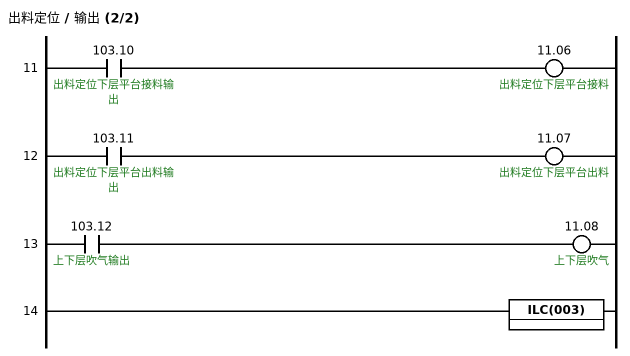
; rung 11
LD 103.10  ; 出料定位下层平台接料输出
OUT 11.06  ; 出料定位下层平台接料
; rung 12
LD 103.11  ; 出料定位下层平台出料输出
OUT 11.07  ; 出料定位下层平台出料
; rung 13
LD 103.12  ; 上下层吹气输出
OUT 11.08  ; 上下层吹气
; rung 14
ILC(003)

### Section END
; rung 0
END(001)

## Program 进出料转移 (cyclic task 3)

### Section Main

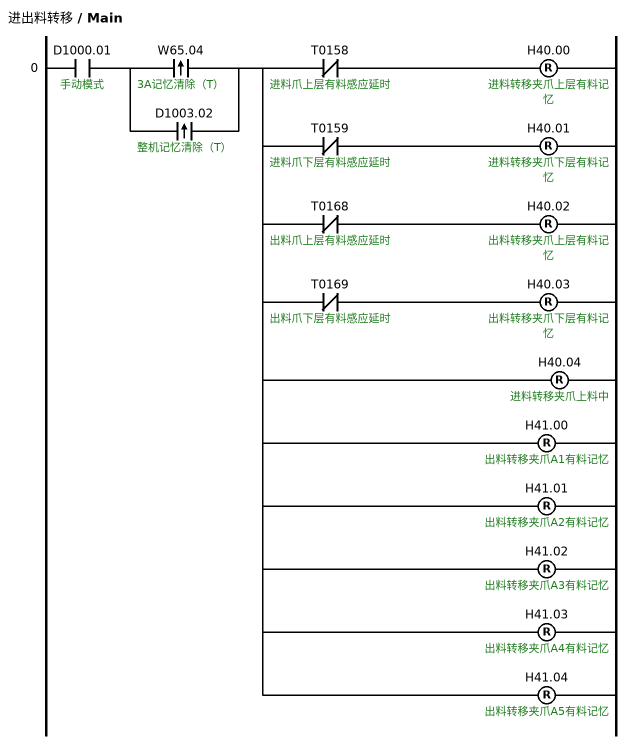
; rung 0
LD D1000.01  ; 手动模式
@LD W65.04  ; 3A记忆清除（T）
@OR D1003.02  ; 整机记忆清除（T）
ANDLD
OUT TR0
ANDNOT T0158  ; 进料爪上层有料感应延时
RSET H40.00  ; 进料转移夹爪上层有料记忆
LD TR0
ANDNOT T0159  ; 进料爪下层有料感应延时
RSET H40.01  ; 进料转移夹爪下层有料记忆
LD TR0
ANDNOT T0168  ; 出料爪上层有料感应延时
RSET H40.02  ; 出料转移夹爪上层有料记忆
LD TR0
ANDNOT T0169  ; 出料爪下层有料感应延时
RSET H40.03  ; 出料转移夹爪下层有料记忆
LD TR0
RSET H40.04  ; 进料转移夹爪上料中
RSET H41.00  ; 出料转移夹爪A1有料记忆
RSET H41.01  ; 出料转移夹爪A2有料记忆
RSET H41.02  ; 出料转移夹爪A3有料记忆
RSET H41.03  ; 出料转移夹爪A4有料记忆
RSET H41.04  ; 出料转移夹爪A5有料记忆

### Section _3ST进出料转移

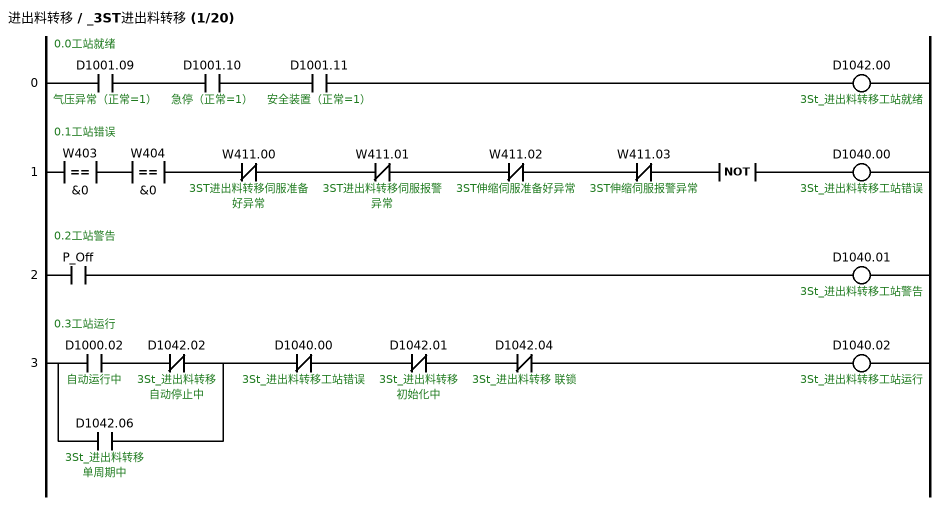
; rung 0: 0.0工站就绪
LD D1001.09  ; 气压异常（正常=1）
AND D1001.10  ; 急停（正常=1）
AND D1001.11  ; 安全装置（正常=1）
OUT D1042.00  ; 3St_进出料转移工站就绪
; rung 1: 0.1工站错误
LD=(300) W403 &0
AND=(300) W404 &0
ANDNOT W411.00  ; 3ST进出料转移伺服准备好异常
ANDNOT W411.01  ; 3ST进出料转移伺服报警异常
ANDNOT W411.02  ; 3ST伸缩伺服准备好异常
ANDNOT W411.03  ; 3ST伸缩伺服报警异常
NOT(520)
OUT D1040.00  ; 3St_进出料转移工站错误
; rung 2: 0.2工站警告
LD P_Off
OUT D1040.01  ; 3St_进出料转移工站警告
; rung 3: 0.3工站运行
LD D1000.02  ; 自动运行中
ANDNOT D1042.02  ; 3St_进出料转移 自动停止中
OR D1042.06  ; 3St_进出料转移 单周期中
ANDNOT D1040.00  ; 3St_进出料转移工站错误
ANDNOT D1042.01  ; 3St_进出料转移 初始化中
ANDNOT D1042.04  ; 3St_进出料转移 联锁
OUT D1040.02  ; 3St_进出料转移工站运行

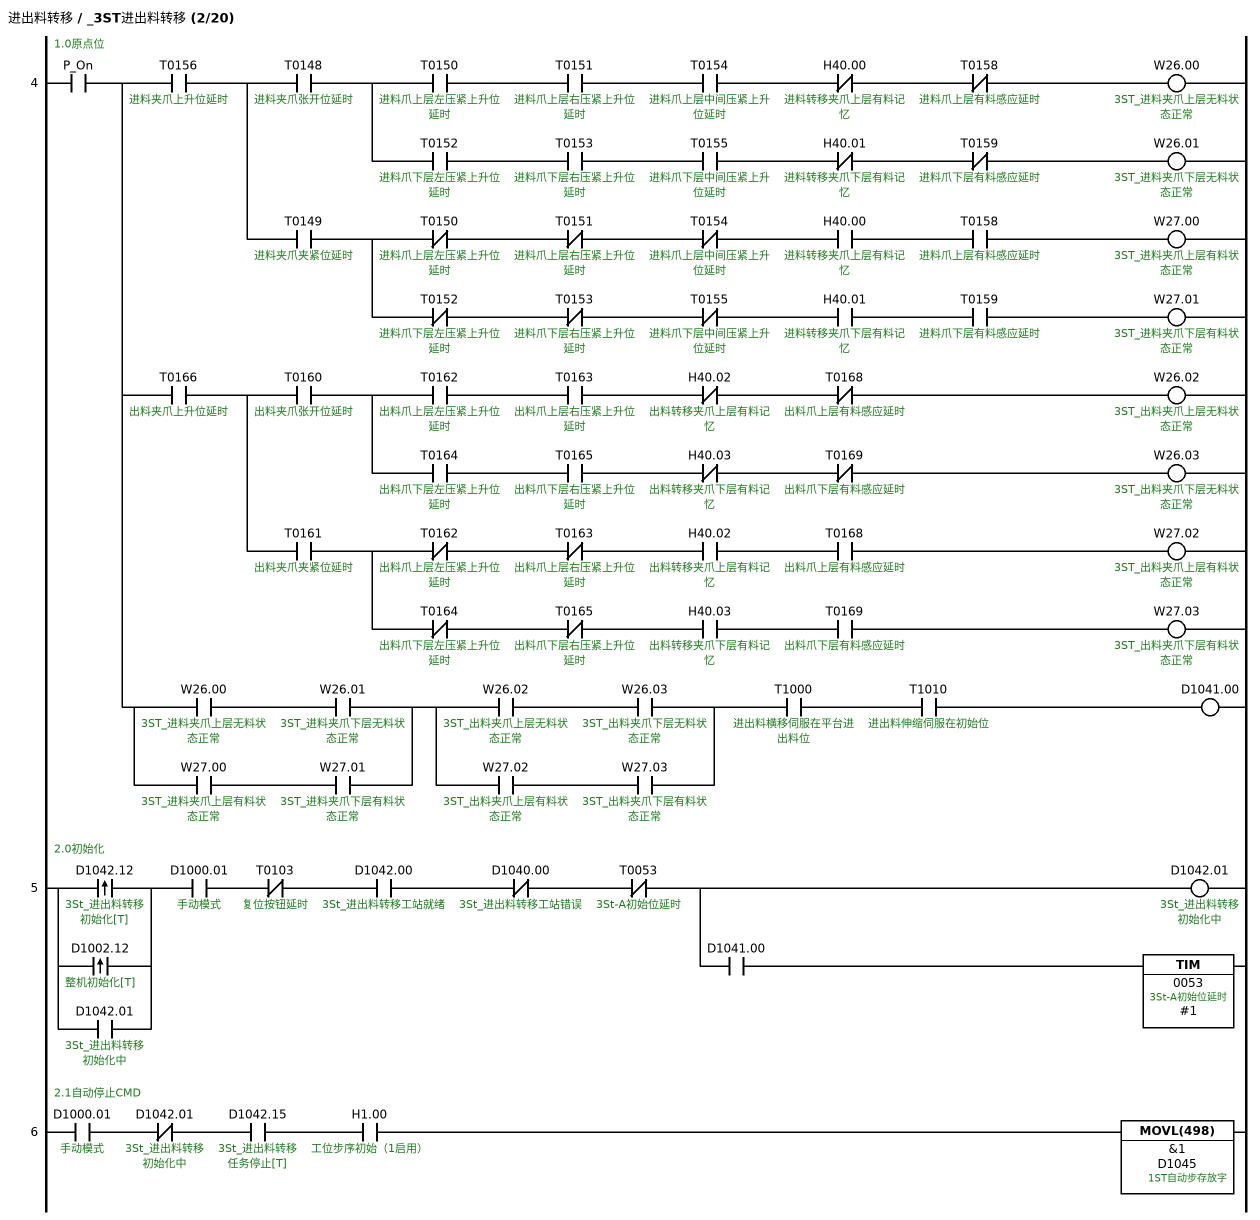
; rung 4: 1.0原点位
LD P_On
OUT TR0
AND T0156  ; 进料夹爪上升位延时
OUT TR1
AND T0148  ; 进料夹爪张开位延时
OUT TR2
AND T0150  ; 进料爪上层左压紧上升位延时
AND T0151  ; 进料爪上层右压紧上升位延时
AND T0154  ; 进料爪上层中间压紧上升位延时
ANDNOT H40.00  ; 进料转移夹爪上层有料记忆
ANDNOT T0158  ; 进料爪上层有料感应延时
OUT W26.00  ; 3ST_进料夹爪上层无料状态正常
LD TR2
AND T0152  ; 进料爪下层左压紧上升位延时
AND T0153  ; 进料爪下层右压紧上升位延时
AND T0155  ; 进料爪下层中间压紧上升位延时
ANDNOT H40.01  ; 进料转移夹爪下层有料记忆
ANDNOT T0159  ; 进料爪下层有料感应延时
OUT W26.01  ; 3ST_进料夹爪下层无料状态正常
LD TR1
AND T0149  ; 进料夹爪夹紧位延时
OUT TR1
ANDNOT T0150  ; 进料爪上层左压紧上升位延时
ANDNOT T0151  ; 进料爪上层右压紧上升位延时
ANDNOT T0154  ; 进料爪上层中间压紧上升位延时
AND H40.00  ; 进料转移夹爪上层有料记忆
AND T0158  ; 进料爪上层有料感应延时
OUT W27.00  ; 3ST_进料夹爪上层有料状态正常
LD TR1
ANDNOT T0152  ; 进料爪下层左压紧上升位延时
ANDNOT T0153  ; 进料爪下层右压紧上升位延时
ANDNOT T0155  ; 进料爪下层中间压紧上升位延时
AND H40.01  ; 进料转移夹爪下层有料记忆
AND T0159  ; 进料爪下层有料感应延时
OUT W27.01  ; 3ST_进料夹爪下层有料状态正常
LD TR0
AND T0166  ; 出料夹爪上升位延时
OUT TR1
AND T0160  ; 出料夹爪张开位延时
OUT TR2
AND T0162  ; 出料爪上层左压紧上升位延时
AND T0163  ; 出料爪上层右压紧上升位延时
ANDNOT H40.02  ; 出料转移夹爪上层有料记忆
ANDNOT T0168  ; 出料爪上层有料感应延时
OUT W26.02  ; 3ST_出料夹爪上层无料状态正常
LD TR2
AND T0164  ; 出料爪下层左压紧上升位延时
AND T0165  ; 出料爪下层右压紧上升位延时
ANDNOT H40.03  ; 出料转移夹爪下层有料记忆
ANDNOT T0169  ; 出料爪下层有料感应延时
OUT W26.03  ; 3ST_出料夹爪下层无料状态正常
LD TR1
AND T0161  ; 出料夹爪夹紧位延时
OUT TR1
ANDNOT T0162  ; 出料爪上层左压紧上升位延时
ANDNOT T0163  ; 出料爪上层右压紧上升位延时
AND H40.02  ; 出料转移夹爪上层有料记忆
AND T0168  ; 出料爪上层有料感应延时
OUT W27.02  ; 3ST_出料夹爪上层有料状态正常
LD TR1
ANDNOT T0164  ; 出料爪下层左压紧上升位延时
ANDNOT T0165  ; 出料爪下层右压紧上升位延时
AND H40.03  ; 出料转移夹爪下层有料记忆
AND T0169  ; 出料爪下层有料感应延时
OUT W27.03  ; 3ST_出料夹爪下层有料状态正常
LD TR0
LD W26.00  ; 3ST_进料夹爪上层无料状态正常
AND W26.01  ; 3ST_进料夹爪下层无料状态正常
LD W27.00  ; 3ST_进料夹爪上层有料状态正常
AND W27.01  ; 3ST_进料夹爪下层有料状态正常
ORLD
ANDLD
LD W26.02  ; 3ST_出料夹爪上层无料状态正常
AND W26.03  ; 3ST_出料夹爪下层无料状态正常
LD W27.02  ; 3ST_出料夹爪上层有料状态正常
AND W27.03  ; 3ST_出料夹爪下层有料状态正常
ORLD
ANDLD
AND T1000  ; 进出料横移伺服在平台进出料位
AND T1010  ; 进出料伸缩伺服在初始位
OUT D1041.00
; rung 5: 2.0初始化
@LD D1042.12  ; 3St_进出料转移 初始化[T]
@OR D1002.12  ; 整机初始化[T]
OR D1042.01  ; 3St_进出料转移 初始化中
AND D1000.01  ; 手动模式
ANDNOT T0103  ; 复位按钮延时
AND D1042.00  ; 3St_进出料转移工站就绪
ANDNOT D1040.00  ; 3St_进出料转移工站错误
ANDNOT T0053  ; 3St-A初始位延时
OUT D1042.01  ; 3St_进出料转移 初始化中
AND D1041.00
TIM 0053 #1  ; 3St-A初始位延时
; rung 6: 2.1自动停止CMD
LD D1000.01  ; 手动模式
ANDNOT D1042.01  ; 3St_进出料转移 初始化中
AND D1042.15  ; 3St_进出料转移 任务停止[T]
AND H1.00  ; 工位步序初始（1启用）
MOVL(498) &1 D1045  ; 1ST自动步存放字

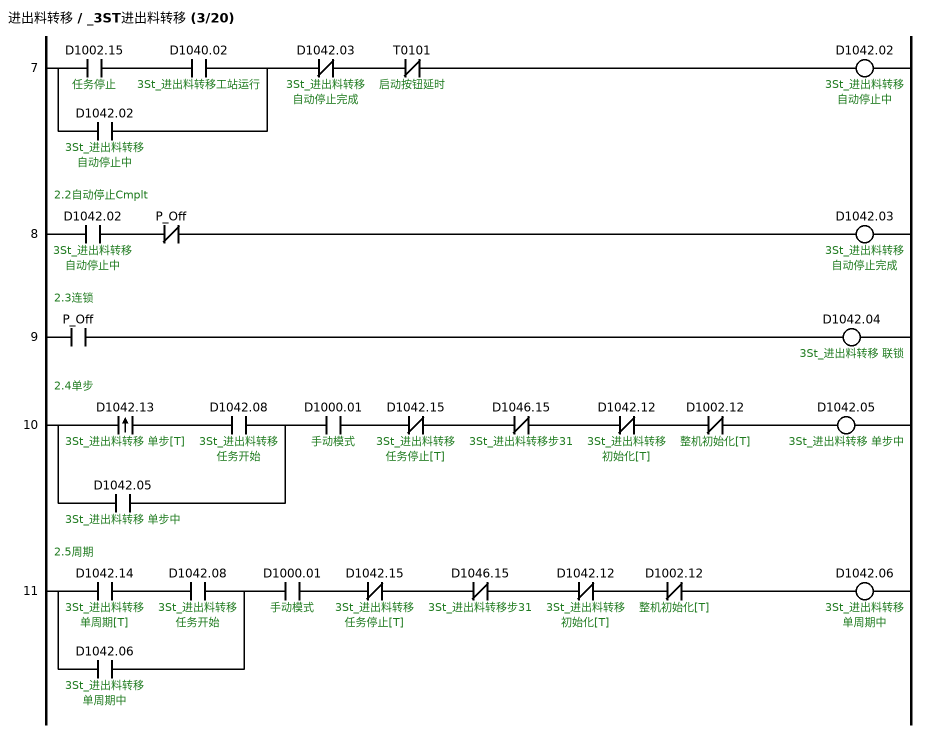
; rung 7
LD D1002.15  ; 任务停止
AND D1040.02  ; 3St_进出料转移工站运行
OR D1042.02  ; 3St_进出料转移 自动停止中
ANDNOT D1042.03  ; 3St_进出料转移 自动停止完成
ANDNOT T0101  ; 启动按钮延时
OUT D1042.02  ; 3St_进出料转移 自动停止中
; rung 8: 2.2自动停止Cmplt
LD D1042.02  ; 3St_进出料转移 自动停止中
ANDNOT P_Off
OUT D1042.03  ; 3St_进出料转移 自动停止完成
; rung 9: 2.3连锁
LD P_Off
OUT D1042.04  ; 3St_进出料转移 联锁
; rung 10: 2.4单步
@LD D1042.13  ; 3St_进出料转移 单步[T]
AND D1042.08  ; 3St_进出料转移 任务开始
OR D1042.05  ; 3St_进出料转移 单步中
AND D1000.01  ; 手动模式
ANDNOT D1042.15  ; 3St_进出料转移 任务停止[T]
ANDNOT D1046.15  ; 3St_进出料转移步31
ANDNOT D1042.12  ; 3St_进出料转移 初始化[T]
ANDNOT D1002.12  ; 整机初始化[T]
OUT D1042.05  ; 3St_进出料转移 单步中
; rung 11: 2.5周期
LD D1042.14  ; 3St_进出料转移 单周期[T]
AND D1042.08  ; 3St_进出料转移 任务开始
OR D1042.06  ; 3St_进出料转移 单周期中
AND D1000.01  ; 手动模式
ANDNOT D1042.15  ; 3St_进出料转移 任务停止[T]
ANDNOT D1046.15  ; 3St_进出料转移步31
ANDNOT D1042.12  ; 3St_进出料转移 初始化[T]
ANDNOT D1002.12  ; 整机初始化[T]
OUT D1042.06  ; 3St_进出料转移 单周期中

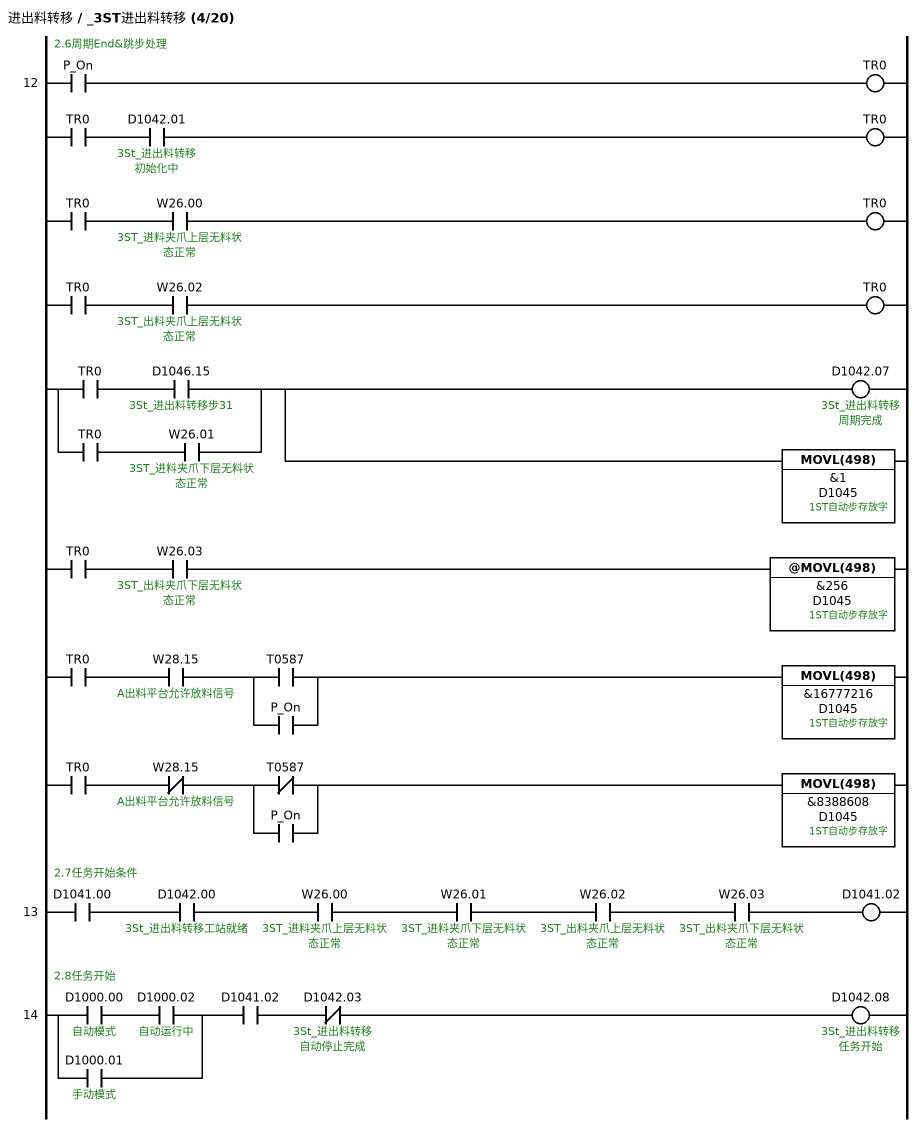
; rung 12: 2.6周期End&跳步处理
LD P_On
OUT TR0
AND D1046.15  ; 3St_进出料转移步31
LD TR0
AND D1042.01  ; 3St_进出料转移 初始化中
OUT TR0
AND W26.01  ; 3ST_进料夹爪下层无料状态正常
ORLD
OUT D1042.07  ; 3St_进出料转移 周期完成
MOVL(498) &1 D1045  ; 1ST自动步存放字
LD TR0
AND W26.00  ; 3ST_进料夹爪上层无料状态正常
OUT TR0
AND W26.03  ; 3ST_出料夹爪下层无料状态正常
@MOVL(498) &256 D1045  ; 1ST自动步存放字  // D1045.08  3ST_A到进料等待位
LD TR0
AND W26.02  ; 3ST_出料夹爪上层无料状态正常
OUT TR0
AND W28.15  ; A出料平台允许放料信号
LD T0587
OR P_On
ANDLD
MOVL(498) &16777216 D1045  ; 1ST自动步存放字  // D1046.08  3ST_A到出料位出料/夹爪下降
LD TR0
ANDNOT W28.15  ; A出料平台允许放料信号
LDNOT T0587
OR P_On
ANDLD
MOVL(498) &8388608 D1045  ; 1ST自动步存放字  // D1046.07  3ST_A到出料等待位
; rung 13: 2.7任务开始条件
LD D1041.00
AND D1042.00  ; 3St_进出料转移工站就绪
AND W26.00  ; 3ST_进料夹爪上层无料状态正常
AND W26.01  ; 3ST_进料夹爪下层无料状态正常
AND W26.02  ; 3ST_出料夹爪上层无料状态正常
AND W26.03  ; 3ST_出料夹爪下层无料状态正常
OUT D1041.02
; rung 14: 2.8任务开始
LD D1000.00  ; 自动模式
AND D1000.02  ; 自动运行中
OR D1000.01  ; 手动模式
AND D1041.02
ANDNOT D1042.03  ; 3St_进出料转移 自动停止完成
OUT D1042.08  ; 3St_进出料转移 任务开始

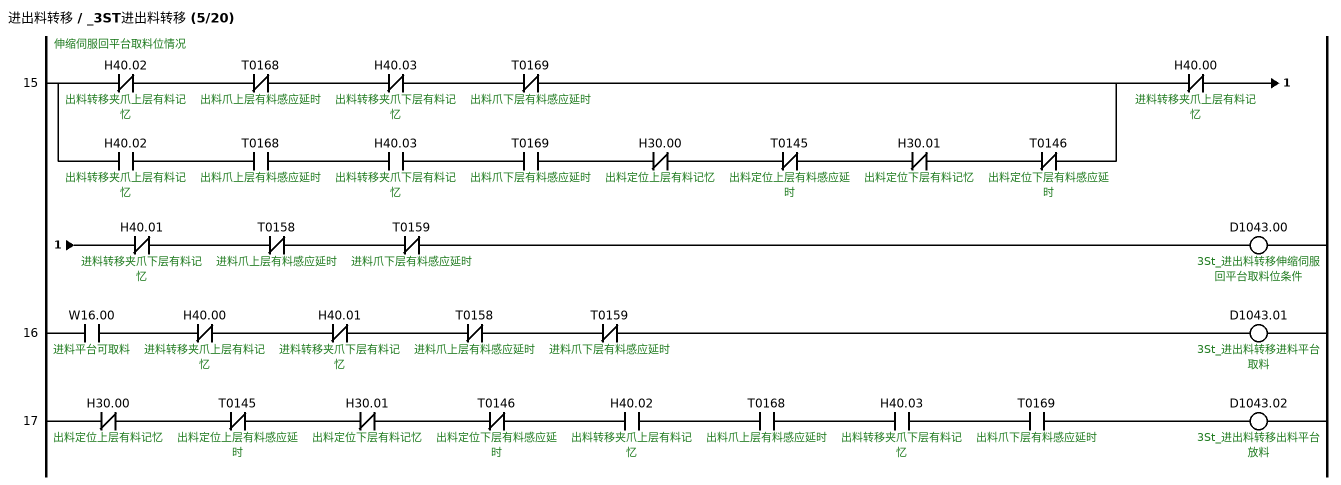
; rung 15: 伸缩伺服回平台取料位情况
LDNOT H40.02  ; 出料转移夹爪上层有料记忆
ANDNOT T0168  ; 出料爪上层有料感应延时
ANDNOT H40.03  ; 出料转移夹爪下层有料记忆
ANDNOT T0169  ; 出料爪下层有料感应延时
LD H40.02  ; 出料转移夹爪上层有料记忆
AND T0168  ; 出料爪上层有料感应延时
AND H40.03  ; 出料转移夹爪下层有料记忆
AND T0169  ; 出料爪下层有料感应延时
ANDNOT H30.00  ; 出料定位上层有料记忆
ANDNOT T0145  ; 出料定位上层有料感应延时
ANDNOT H30.01  ; 出料定位下层有料记忆
ANDNOT T0146  ; 出料定位下层有料感应延时
ORLD
ANDNOT H40.00  ; 进料转移夹爪上层有料记忆
ANDNOT H40.01  ; 进料转移夹爪下层有料记忆
ANDNOT T0158  ; 进料爪上层有料感应延时
ANDNOT T0159  ; 进料爪下层有料感应延时
OUT D1043.00  ; 3St_进出料转移伸缩伺服回平台取料位条件
; rung 16
LD W16.00  ; 进料平台可取料
ANDNOT H40.00  ; 进料转移夹爪上层有料记忆
ANDNOT H40.01  ; 进料转移夹爪下层有料记忆
ANDNOT T0158  ; 进料爪上层有料感应延时
ANDNOT T0159  ; 进料爪下层有料感应延时
OUT D1043.01  ; 3St_进出料转移进料平台取料
; rung 17
LDNOT H30.00  ; 出料定位上层有料记忆
ANDNOT T0145  ; 出料定位上层有料感应延时
ANDNOT H30.01  ; 出料定位下层有料记忆
ANDNOT T0146  ; 出料定位下层有料感应延时
AND H40.02  ; 出料转移夹爪上层有料记忆
AND T0168  ; 出料爪上层有料感应延时
AND H40.03  ; 出料转移夹爪下层有料记忆
AND T0169  ; 出料爪下层有料感应延时
OUT D1043.02  ; 3St_进出料转移出料平台放料

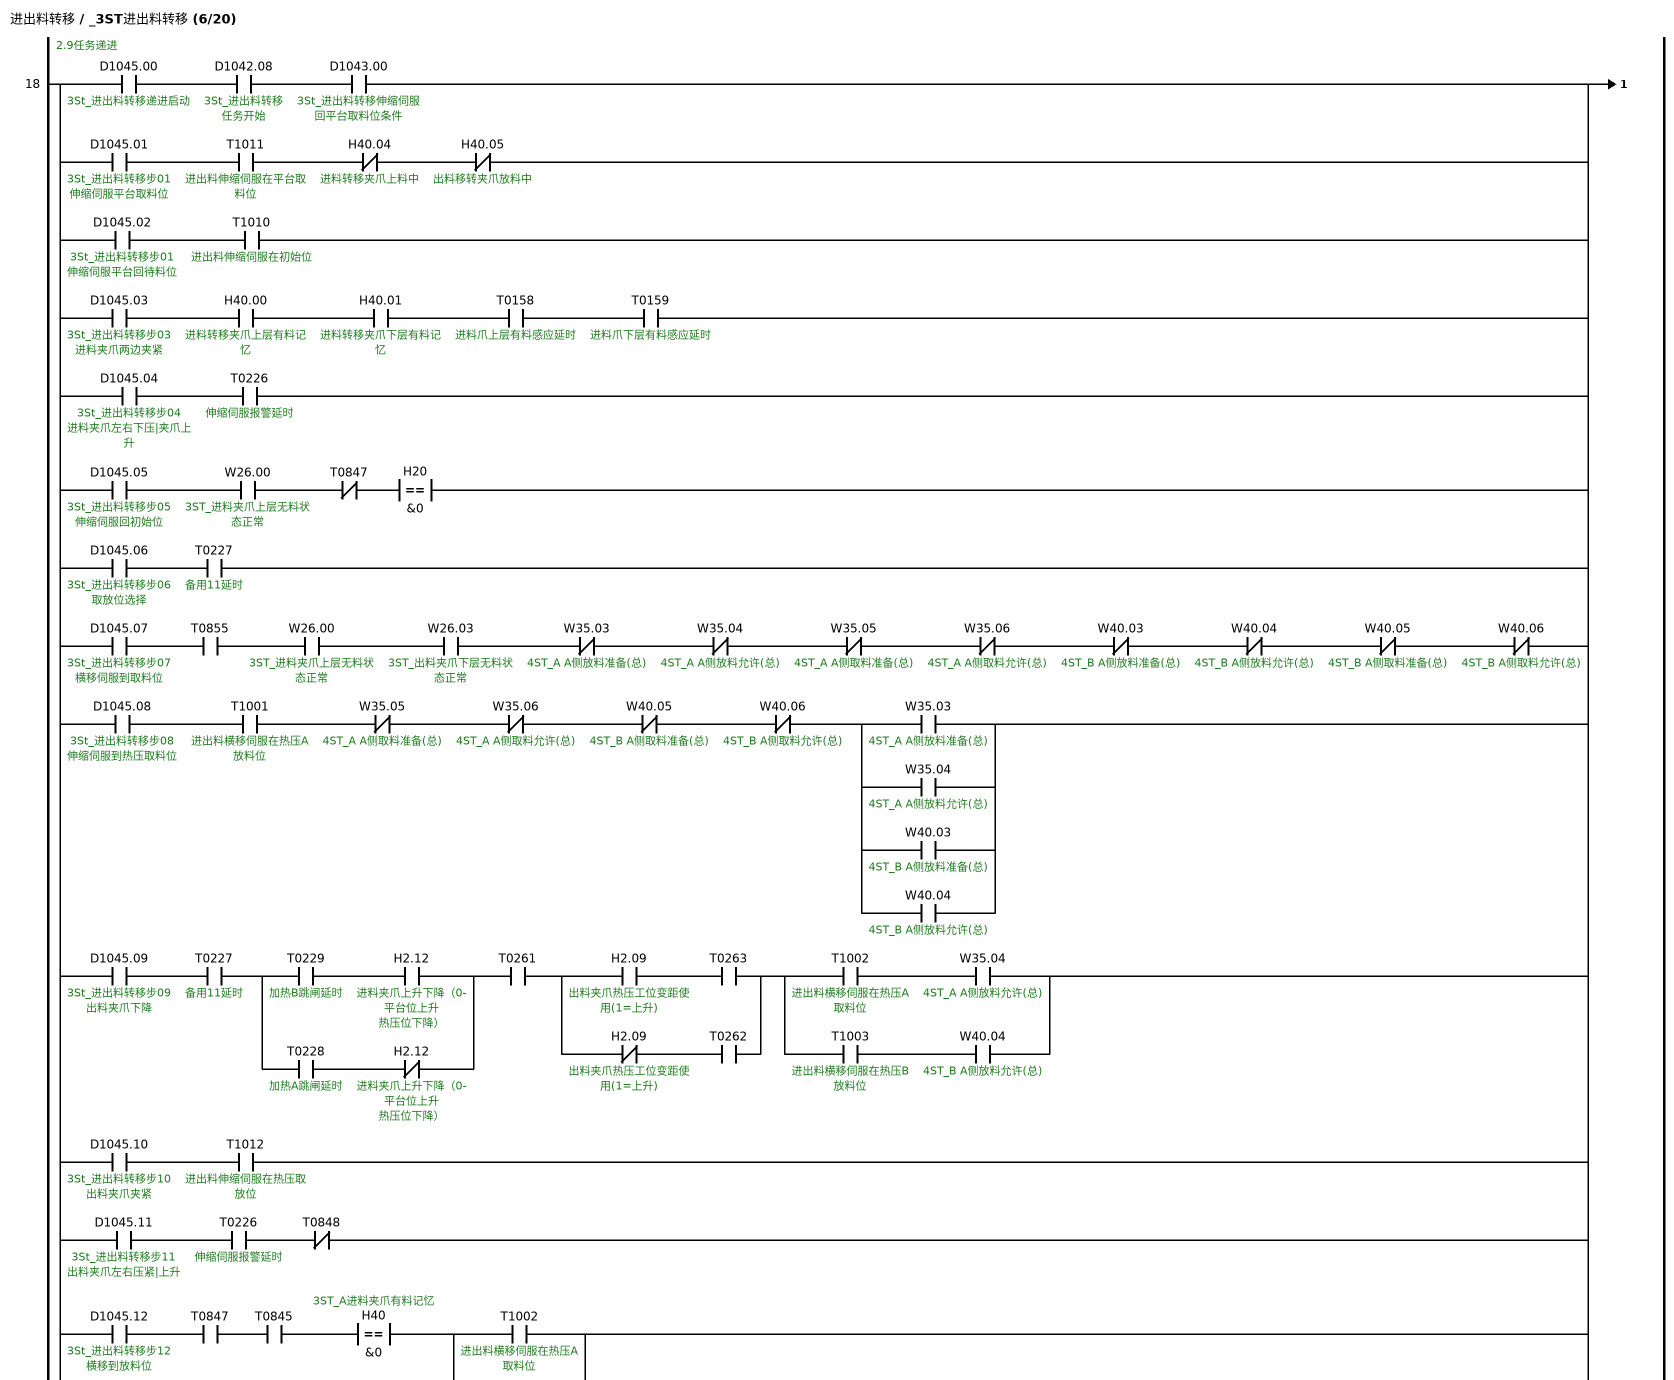

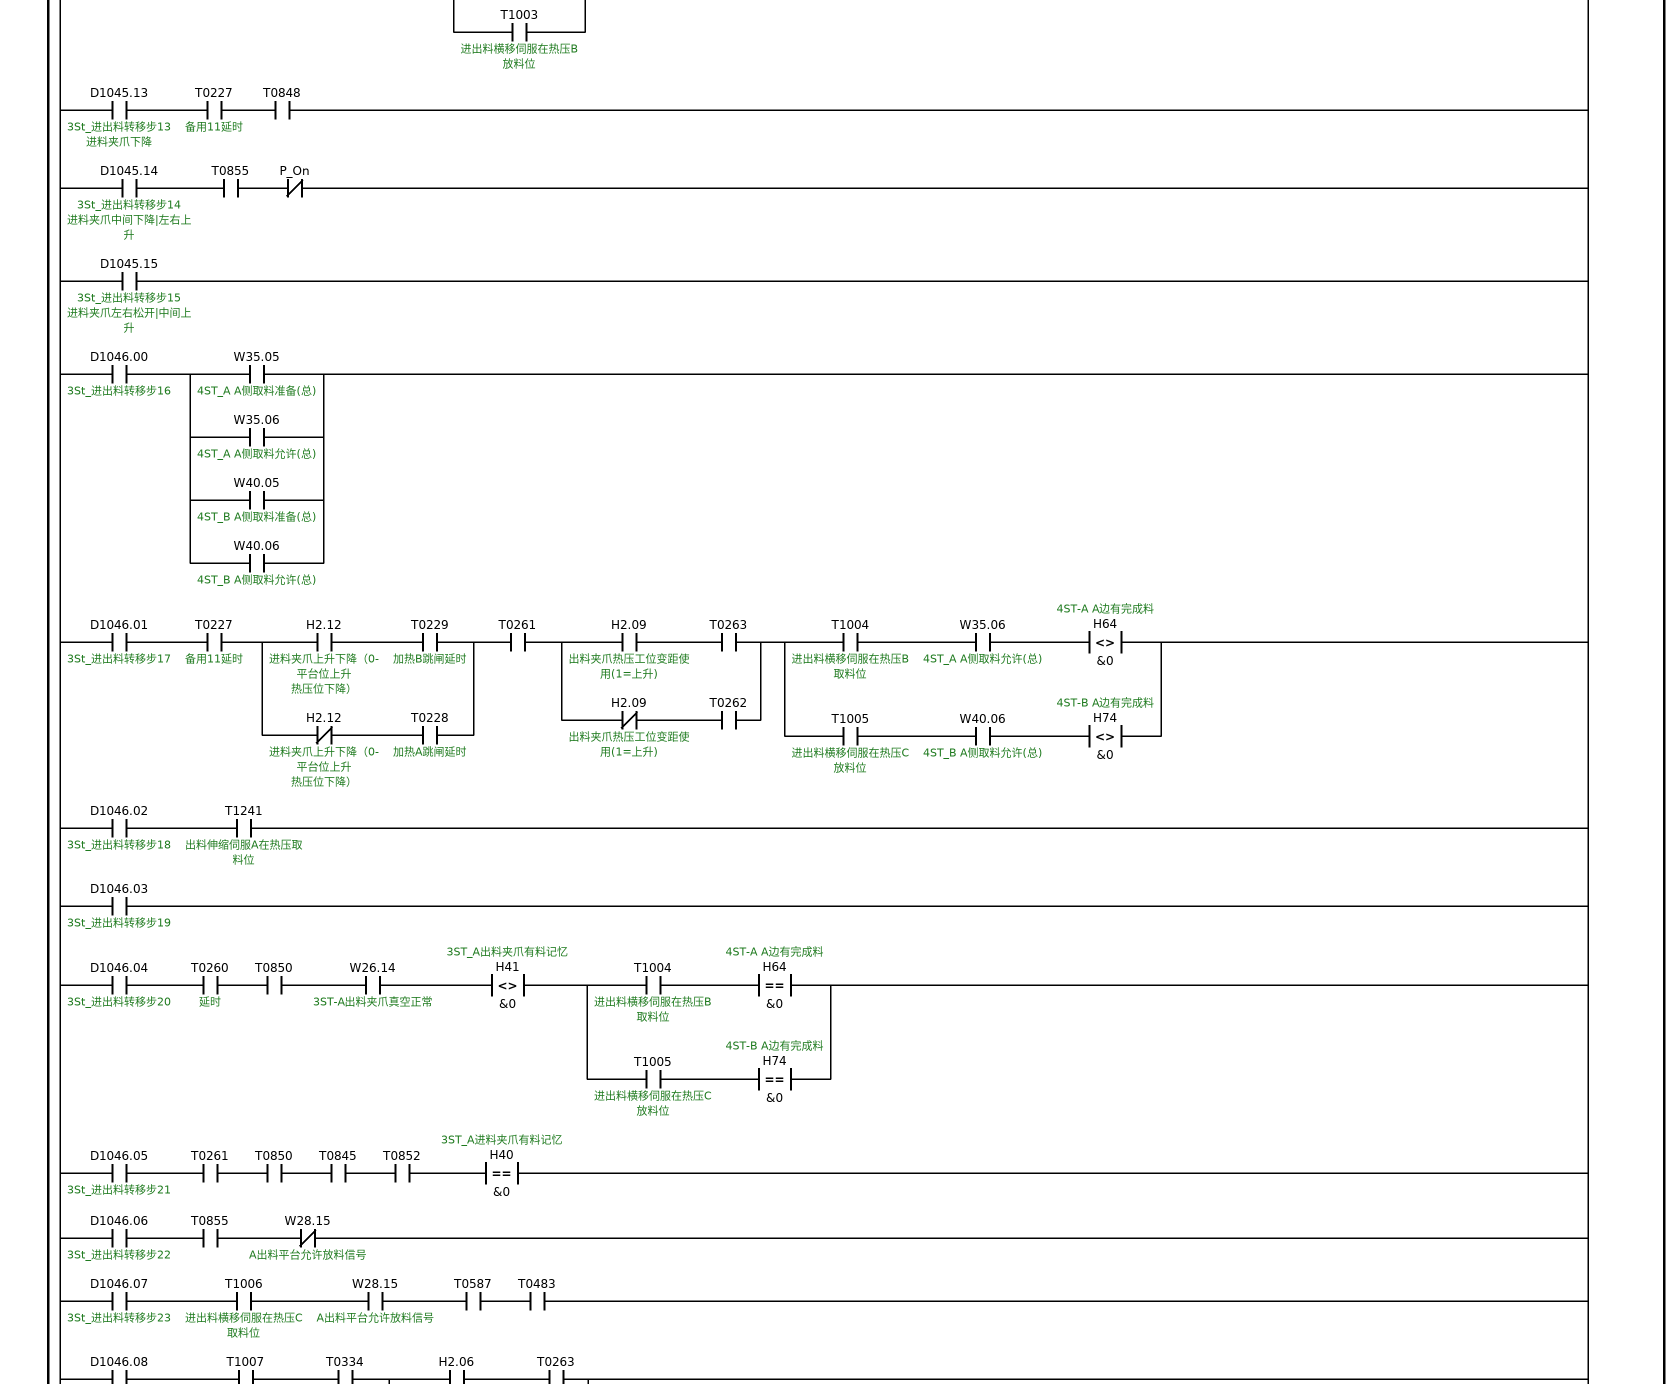

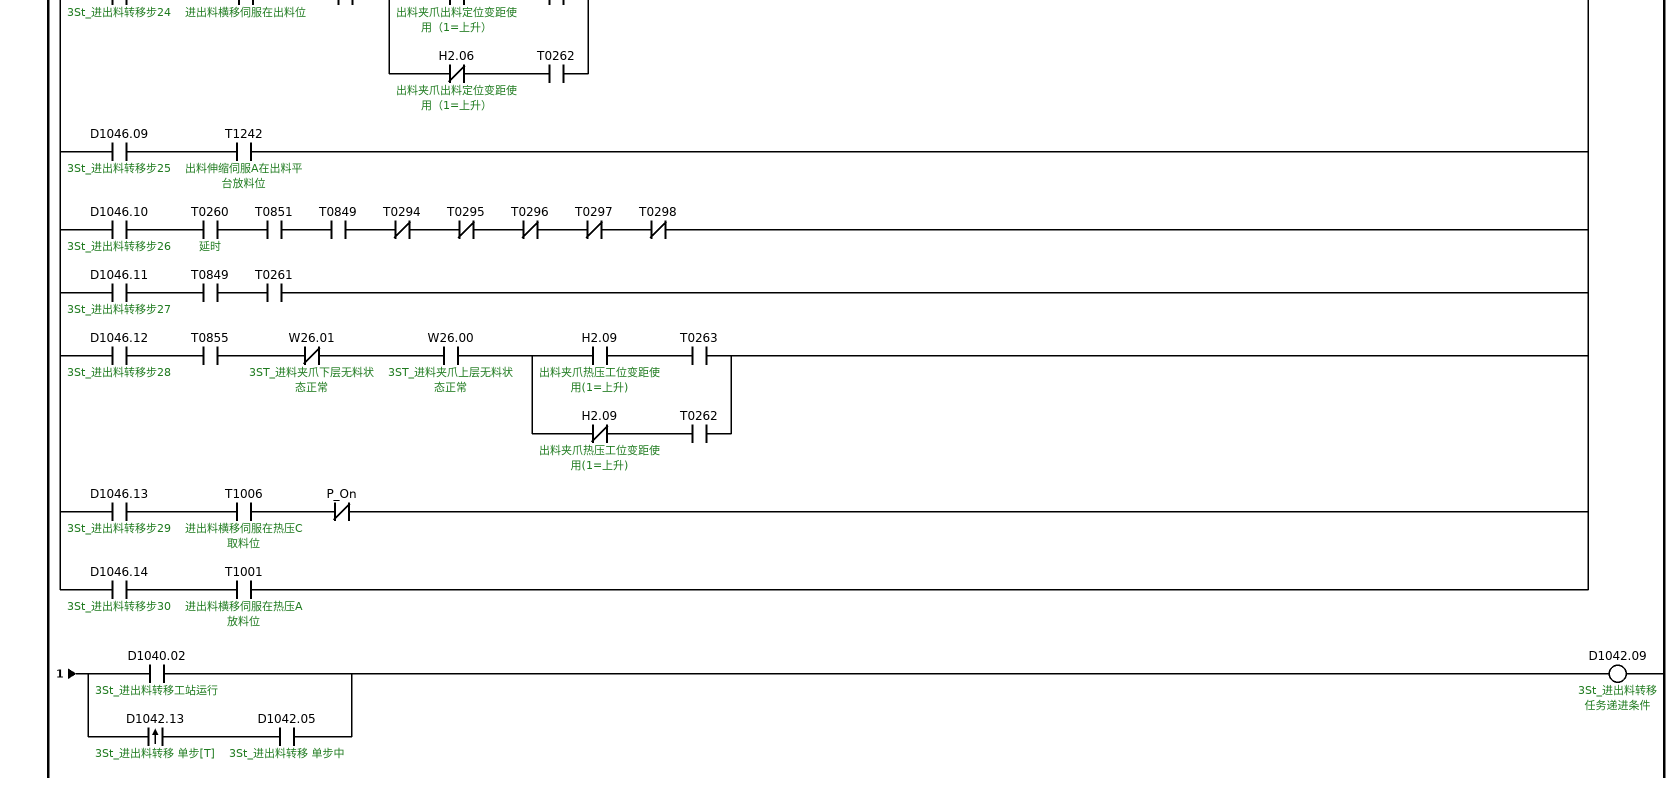
; rung 18: 2.9任务递进
LD D1045.00  ; 3St_进出料转移递进启动
AND D1042.08  ; 3St_进出料转移 任务开始
AND D1043.00  ; 3St_进出料转移伸缩伺服回平台取料位条件
LD D1045.01  ; 3St_进出料转移步01 伸缩伺服平台取料位  // 进料平台可取料则跳入取料步；出料平台可放料则跳入放料步；取放料完成后跳入D1045.02步
AND T1011  ; 进出料伸缩伺服在平台取料位
ANDNOT H40.04  ; 进料转移夹爪上料中
ANDNOT H40.05  ; 出料移转夹爪放料中
ORLD
LD D1045.02  ; 3St_进出料转移步01 伸缩伺服平台回待料位
AND T1010  ; 进出料伸缩伺服在初始位
ORLD
LD D1045.03  ; 3St_进出料转移步03 进料夹爪两边夹紧  // 进料
AND H40.00  ; 进料转移夹爪上层有料记忆
AND H40.01  ; 进料转移夹爪下层有料记忆
AND T0158  ; 进料爪上层有料感应延时
AND T0159  ; 进料爪下层有料感应延时
ORLD
LD D1045.04  ; 3St_进出料转移步04 进料夹爪左右下压|夹爪上升
AND T0226  ; 伸缩伺服报警延时
ORLD
LD D1045.05  ; 3St_进出料转移步05 伸缩伺服回初始位
AND W26.00  ; 3ST_进料夹爪上层无料状态正常
ANDNOT T0847
AND=(300) H20 &0
ORLD
LD D1045.06  ; 3St_进出料转移步06 取放位选择
AND T0227  ; 备用11延时
ORLD
LD D1045.07  ; 3St_进出料转移步07 横移伺服到取料位
AND T0855
AND W26.00  ; 3ST_进料夹爪上层无料状态正常
AND W26.03  ; 3ST_出料夹爪下层无料状态正常
ANDNOT W35.03  ; 4ST_A A侧放料准备(总)
ANDNOT W35.04  ; 4ST_A A侧放料允许(总)
ANDNOT W35.05  ; 4ST_A A侧取料准备(总)
ANDNOT W35.06  ; 4ST_A A侧取料允许(总)
ANDNOT W40.03  ; 4ST_B A侧放料准备(总)
ANDNOT W40.04  ; 4ST_B A侧放料允许(总)
ANDNOT W40.05  ; 4ST_B A侧取料准备(总)
ANDNOT W40.06  ; 4ST_B A侧取料允许(总)
ORLD
LD D1045.08  ; 3St_进出料转移步08 伸缩伺服到热压取料位
AND T1001  ; 进出料横移伺服在热压A放料位
ANDNOT W35.05  ; 4ST_A A侧取料准备(总)
ANDNOT W35.06  ; 4ST_A A侧取料允许(总)
ANDNOT W40.05  ; 4ST_B A侧取料准备(总)
ANDNOT W40.06  ; 4ST_B A侧取料允许(总)
LD W35.03  ; 4ST_A A侧放料准备(总)
OR W35.04  ; 4ST_A A侧放料允许(总)
OR W40.03  ; 4ST_B A侧放料准备(总)
OR W40.04  ; 4ST_B A侧放料允许(总)
ANDLD
ORLD
LD D1045.09  ; 3St_进出料转移步09 出料夹爪下降
AND T0227  ; 备用11延时
LD T0229  ; 加热B跳闸延时
AND H2.12  ; 进料夹爪上升下降（0-平台位上升  热压位下降）
LD T0228  ; 加热A跳闸延时
ANDNOT H2.12  ; 进料夹爪上升下降（0-平台位上升  热压位下降）
ORLD
ANDLD
AND T0261
LD H2.09  ; 出料夹爪热压工位变距使用(1=上升)
AND T0263
LDNOT H2.09  ; 出料夹爪热压工位变距使用(1=上升)
AND T0262
ORLD
ANDLD
LD T1002  ; 进出料横移伺服在热压A取料位
AND W35.04  ; 4ST_A A侧放料允许(总)
LD T1003  ; 进出料横移伺服在热压B放料位
AND W40.04  ; 4ST_B A侧放料允许(总)
ORLD
ANDLD
ORLD
LD D1045.10  ; 3St_进出料转移步10 出料夹爪夹紧
AND T1012  ; 进出料伸缩伺服在热压取放位
ORLD
LD D1045.11  ; 3St_进出料转移步11 出料夹爪左右压紧|上升
AND T0226  ; 伸缩伺服报警延时
ANDNOT T0848
ORLD
LD D1045.12  ; 3St_进出料转移步12 横移到放料位
AND T0847
AND T0845
AND=(300) H40 &0  ; 3ST_A进料夹爪有料记忆
LD T1002  ; 进出料横移伺服在热压A取料位
OR T1003  ; 进出料横移伺服在热压B放料位
ANDLD
ORLD
LD D1045.13  ; 3St_进出料转移步13 进料夹爪下降
AND T0227  ; 备用11延时
AND T0848
ORLD
LD D1045.14  ; 3St_进出料转移步14 进料夹爪中间下降|左右上升
AND T0855
ANDNOT P_On
ORLD
OR D1045.15  ; 3St_进出料转移步15 进料夹爪左右松开|中间上升
LD D1046.00  ; 3St_进出料转移步16
LD W35.05  ; 4ST_A A侧取料准备(总)
OR W35.06  ; 4ST_A A侧取料允许(总)
OR W40.05  ; 4ST_B A侧取料准备(总)
OR W40.06  ; 4ST_B A侧取料允许(总)
ANDLD
ORLD
LD D1046.01  ; 3St_进出料转移步17
AND T0227  ; 备用11延时
LD H2.12  ; 进料夹爪上升下降（0-平台位上升  热压位下降）
AND T0229  ; 加热B跳闸延时
LDNOT H2.12  ; 进料夹爪上升下降（0-平台位上升  热压位下降）
AND T0228  ; 加热A跳闸延时
ORLD
ANDLD
AND T0261
LD H2.09  ; 出料夹爪热压工位变距使用(1=上升)
AND T0263
LDNOT H2.09  ; 出料夹爪热压工位变距使用(1=上升)
AND T0262
ORLD
ANDLD
LD T1004  ; 进出料横移伺服在热压B取料位
AND W35.06  ; 4ST_A A侧取料允许(总)
AND<>(305) H64 &0  ; 4ST-A A边有完成料
LD T1005  ; 进出料横移伺服在热压C放料位
AND W40.06  ; 4ST_B A侧取料允许(总)
AND<>(305) H74 &0  ; 4ST-B A边有完成料
ORLD
ANDLD
ORLD
LD D1046.02  ; 3St_进出料转移步18
AND T1241  ; 出料伸缩伺服A在热压取料位
ORLD
OR D1046.03  ; 3St_进出料转移步19
LD D1046.04  ; 3St_进出料转移步20
AND T0260  ; 延时
AND T0850
AND W26.14  ; 3ST-A出料夹爪真空正常
AND<>(305) H41 &0  ; 3ST_A出料夹爪有料记忆
LD T1004  ; 进出料横移伺服在热压B取料位
AND=(300) H64 &0  ; 4ST-A A边有完成料
LD T1005  ; 进出料横移伺服在热压C放料位
AND=(300) H74 &0  ; 4ST-B A边有完成料
ORLD
ANDLD
ORLD
LD D1046.05  ; 3St_进出料转移步21
AND T0261
AND T0850
AND T0845
AND T0852
AND=(300) H40 &0  ; 3ST_A进料夹爪有料记忆
ORLD
LD D1046.06  ; 3St_进出料转移步22
AND T0855
ANDNOT W28.15  ; A出料平台允许放料信号
ORLD
LD D1046.07  ; 3St_进出料转移步23
AND T1006  ; 进出料横移伺服在热压C取料位
AND W28.15  ; A出料平台允许放料信号
AND T0587
AND T0483
ORLD
LD D1046.08  ; 3St_进出料转移步24
AND T1007  ; 进出料横移伺服在出料位
AND T0334
LD H2.06  ; 出料夹爪出料定位变距使用（1=上升）
AND T0263
LDNOT H2.06  ; 出料夹爪出料定位变距使用（1=上升）
AND T0262
ORLD
ANDLD
ORLD
LD D1046.09  ; 3St_进出料转移步25
AND T1242  ; 出料伸缩伺服A在出料平台放料位
ORLD
LD D1046.10  ; 3St_进出料转移步26
AND T0260  ; 延时
AND T0851
AND T0849
ANDNOT T0294
ANDNOT T0295
ANDNOT T0296
ANDNOT T0297
ANDNOT T0298
ORLD
LD D1046.11  ; 3St_进出料转移步27
AND T0849
AND T0261
ORLD
LD D1046.12  ; 3St_进出料转移步28
AND T0855
ANDNOT W26.01  ; 3ST_进料夹爪下层无料状态正常
AND W26.00  ; 3ST_进料夹爪上层无料状态正常
LD H2.09  ; 出料夹爪热压工位变距使用(1=上升)
AND T0263
LDNOT H2.09  ; 出料夹爪热压工位变距使用(1=上升)
AND T0262
ORLD
ANDLD
ORLD
LD D1046.13  ; 3St_进出料转移步29
AND T1006  ; 进出料横移伺服在热压C取料位
ANDNOT P_On
ORLD
LD D1046.14  ; 3St_进出料转移步30
AND T1001  ; 进出料横移伺服在热压A放料位
ORLD
LD D1040.02  ; 3St_进出料转移工站运行
@LD D1042.13  ; 3St_进出料转移 单步[T]
AND D1042.05  ; 3St_进出料转移 单步中
ORLD
ANDLD
OUT D1042.09  ; 3St_进出料转移 任务递进条件

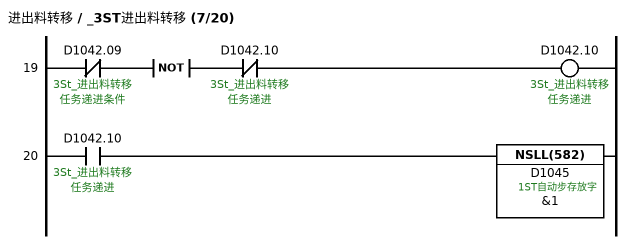
; rung 19
LDNOT D1042.09  ; 3St_进出料转移 任务递进条件
NOT(520)
ANDNOT D1042.10  ; 3St_进出料转移 任务递进
OUT D1042.10  ; 3St_进出料转移 任务递进
; rung 20
LD D1042.10  ; 3St_进出料转移 任务递进
NSLL(582) D1045 &1  ; 1ST自动步存放字

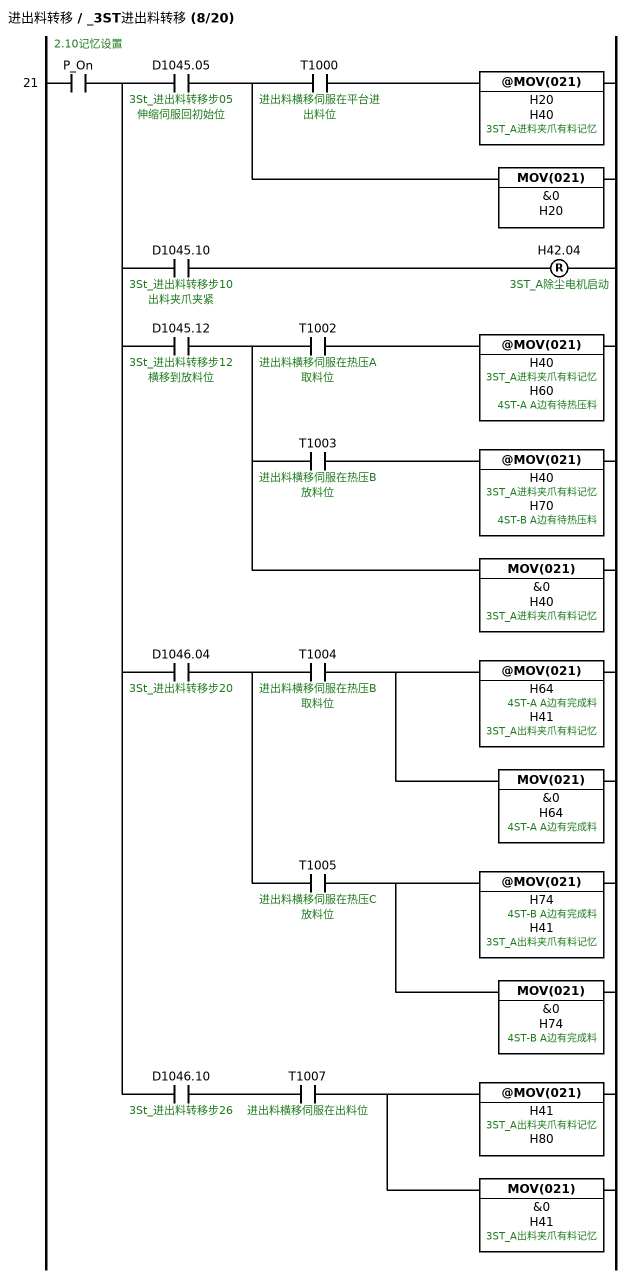
; rung 21: 2.10记忆设置
LD P_On
OUT TR0
AND D1045.05  ; 3St_进出料转移步05 伸缩伺服回初始位
OUT TR1
AND T1000  ; 进出料横移伺服在平台进出料位
@MOV(021) H20 H40  ; 3ST_A进料夹爪有料记忆
LD TR1
MOV(021) &0 H20
LD TR0
AND D1045.10  ; 3St_进出料转移步10 出料夹爪夹紧
RSET H42.04  ; 3ST_A除尘电机启动
LD TR0
AND D1045.12  ; 3St_进出料转移步12 横移到放料位
OUT TR1
AND T1002  ; 进出料横移伺服在热压A取料位
@MOV(021) H40 H60  ; 3ST_A进料夹爪有料记忆, 4ST-A A边有待热压料
LD TR1
AND T1003  ; 进出料横移伺服在热压B放料位
@MOV(021) H40 H70  ; 3ST_A进料夹爪有料记忆, 4ST-B A边有待热压料
LD TR1
MOV(021) &0 H40  ; 3ST_A进料夹爪有料记忆
LD TR0
AND D1046.04  ; 3St_进出料转移步20
OUT TR1
AND T1004  ; 进出料横移伺服在热压B取料位
@MOV(021) H64 H41  ; 4ST-A A边有完成料, 3ST_A出料夹爪有料记忆
MOV(021) &0 H64  ; 4ST-A A边有完成料
LD TR1
AND T1005  ; 进出料横移伺服在热压C放料位
@MOV(021) H74 H41  ; 4ST-B A边有完成料, 3ST_A出料夹爪有料记忆
MOV(021) &0 H74  ; 4ST-B A边有完成料
LD TR0
AND D1046.10  ; 3St_进出料转移步26
AND T1007  ; 进出料横移伺服在出料位
@MOV(021) H41 H80  ; 3ST_A出料夹爪有料记忆
MOV(021) &0 H41  ; 3ST_A出料夹爪有料记忆

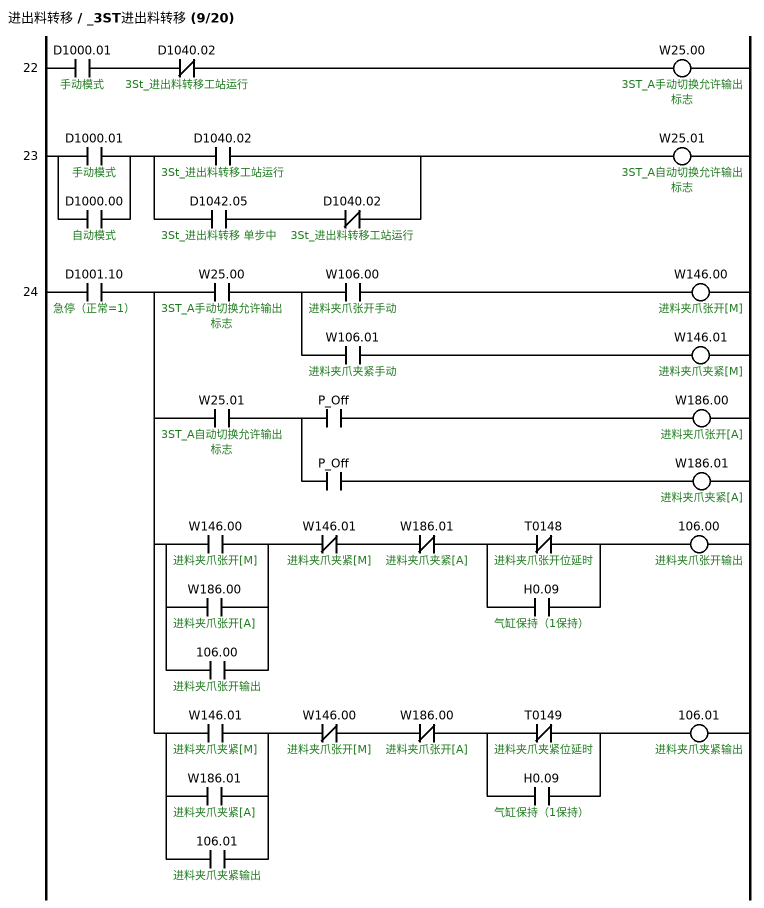
; rung 22
LD D1000.01  ; 手动模式
ANDNOT D1040.02  ; 3St_进出料转移工站运行
OUT W25.00  ; 3ST_A手动切换允许输出标志
; rung 23
LD D1000.01  ; 手动模式
OR D1000.00  ; 自动模式
LD D1040.02  ; 3St_进出料转移工站运行
LD D1042.05  ; 3St_进出料转移 单步中
ANDNOT D1040.02  ; 3St_进出料转移工站运行
ORLD
ANDLD
OUT W25.01  ; 3ST_A自动切换允许输出标志
; rung 24
LD D1001.10  ; 急停（正常=1）
OUT TR0
AND W25.00  ; 3ST_A手动切换允许输出标志
OUT TR1
AND W106.00  ; 进料夹爪张开手动
OUT W146.00  ; 进料夹爪张开[M]
LD TR1
AND W106.01  ; 进料夹爪夹紧手动
OUT W146.01  ; 进料夹爪夹紧[M]
LD TR0
AND W25.01  ; 3ST_A自动切换允许输出标志
OUT TR1
AND P_Off
OUT W186.00  ; 进料夹爪张开[A]
LD TR1
AND P_Off
OUT W186.01  ; 进料夹爪夹紧[A]
LD TR0
LD W146.00  ; 进料夹爪张开[M]
OR W186.00  ; 进料夹爪张开[A]
OR 106.00  ; 进料夹爪张开输出
ANDLD
ANDNOT W146.01  ; 进料夹爪夹紧[M]
ANDNOT W186.01  ; 进料夹爪夹紧[A]
LDNOT T0148  ; 进料夹爪张开位延时
OR H0.09  ; 气缸保持（1保持）
ANDLD
OUT 106.00  ; 进料夹爪张开输出
LD TR0
LD W146.01  ; 进料夹爪夹紧[M]
OR W186.01  ; 进料夹爪夹紧[A]
OR 106.01  ; 进料夹爪夹紧输出
ANDLD
ANDNOT W146.00  ; 进料夹爪张开[M]
ANDNOT W186.00  ; 进料夹爪张开[A]
LDNOT T0149  ; 进料夹爪夹紧位延时
OR H0.09  ; 气缸保持（1保持）
ANDLD
OUT 106.01  ; 进料夹爪夹紧输出

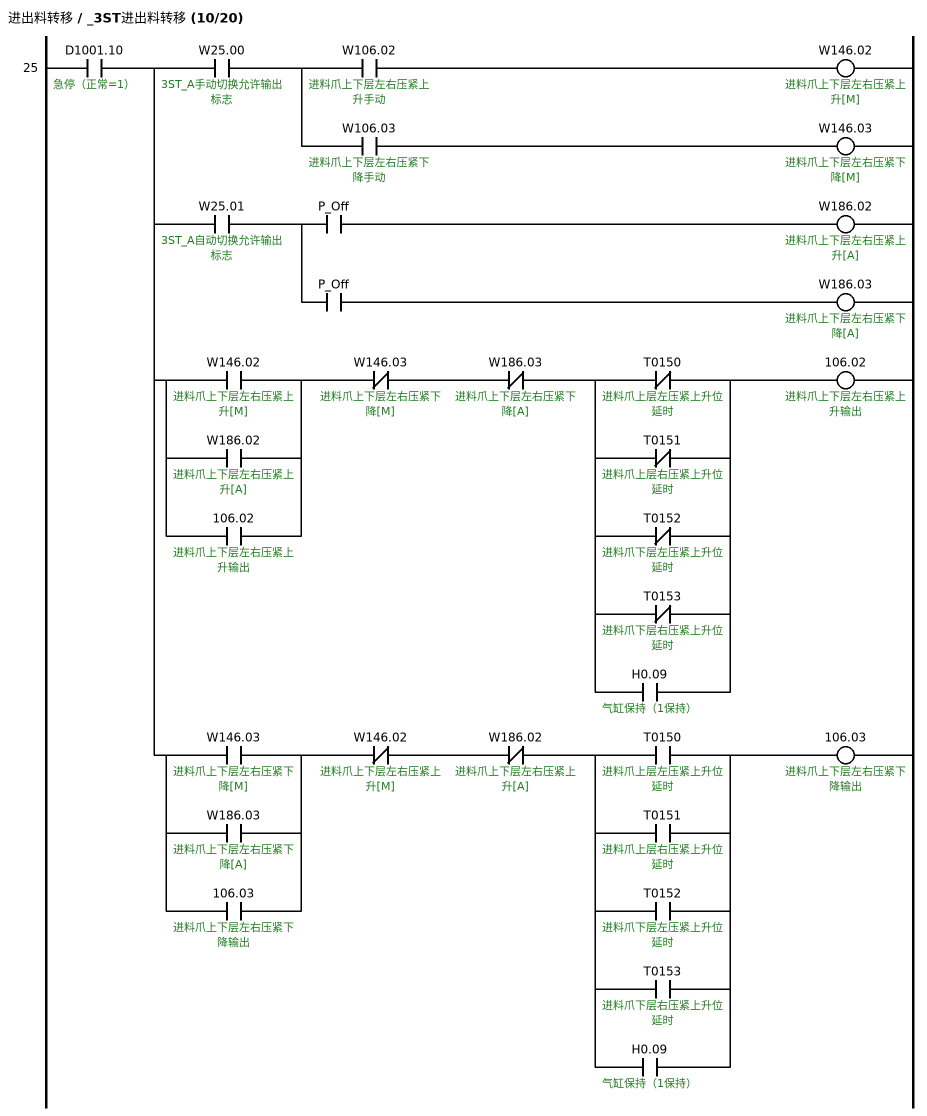
; rung 25
LD D1001.10  ; 急停（正常=1）
OUT TR0
AND W25.00  ; 3ST_A手动切换允许输出标志
OUT TR1
AND W106.02  ; 进料爪上下层左右压紧上升手动
OUT W146.02  ; 进料爪上下层左右压紧上升[M]
LD TR1
AND W106.03  ; 进料爪上下层左右压紧下降手动
OUT W146.03  ; 进料爪上下层左右压紧下降[M]
LD TR0
AND W25.01  ; 3ST_A自动切换允许输出标志
OUT TR1
AND P_Off
OUT W186.02  ; 进料爪上下层左右压紧上升[A]
LD TR1
AND P_Off
OUT W186.03  ; 进料爪上下层左右压紧下降[A]
LD TR0
LD W146.02  ; 进料爪上下层左右压紧上升[M]
OR W186.02  ; 进料爪上下层左右压紧上升[A]
OR 106.02  ; 进料爪上下层左右压紧上升输出
ANDLD
ANDNOT W146.03  ; 进料爪上下层左右压紧下降[M]
ANDNOT W186.03  ; 进料爪上下层左右压紧下降[A]
LDNOT T0150  ; 进料爪上层左压紧上升位延时
ORNOT T0151  ; 进料爪上层右压紧上升位延时
ORNOT T0152  ; 进料爪下层左压紧上升位延时
ORNOT T0153  ; 进料爪下层右压紧上升位延时
OR H0.09  ; 气缸保持（1保持）
ANDLD
OUT 106.02  ; 进料爪上下层左右压紧上升输出
LD TR0
LD W146.03  ; 进料爪上下层左右压紧下降[M]
OR W186.03  ; 进料爪上下层左右压紧下降[A]
OR 106.03  ; 进料爪上下层左右压紧下降输出
ANDLD
ANDNOT W146.02  ; 进料爪上下层左右压紧上升[M]
ANDNOT W186.02  ; 进料爪上下层左右压紧上升[A]
LD T0150  ; 进料爪上层左压紧上升位延时
OR T0151  ; 进料爪上层右压紧上升位延时
OR T0152  ; 进料爪下层左压紧上升位延时
OR T0153  ; 进料爪下层右压紧上升位延时
OR H0.09  ; 气缸保持（1保持）
ANDLD
OUT 106.03  ; 进料爪上下层左右压紧下降输出

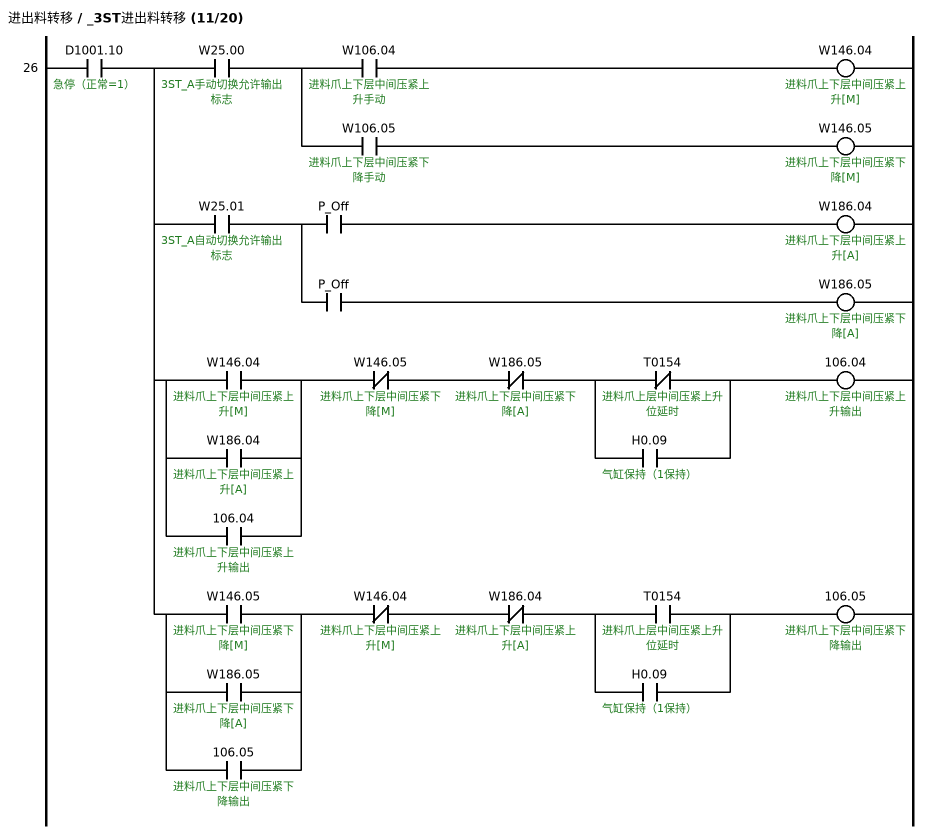
; rung 26
LD D1001.10  ; 急停（正常=1）
OUT TR0
AND W25.00  ; 3ST_A手动切换允许输出标志
OUT TR1
AND W106.04  ; 进料爪上下层中间压紧上升手动
OUT W146.04  ; 进料爪上下层中间压紧上升[M]
LD TR1
AND W106.05  ; 进料爪上下层中间压紧下降手动
OUT W146.05  ; 进料爪上下层中间压紧下降[M]
LD TR0
AND W25.01  ; 3ST_A自动切换允许输出标志
OUT TR1
AND P_Off
OUT W186.04  ; 进料爪上下层中间压紧上升[A]
LD TR1
AND P_Off
OUT W186.05  ; 进料爪上下层中间压紧下降[A]
LD TR0
LD W146.04  ; 进料爪上下层中间压紧上升[M]
OR W186.04  ; 进料爪上下层中间压紧上升[A]
OR 106.04  ; 进料爪上下层中间压紧上升输出
ANDLD
ANDNOT W146.05  ; 进料爪上下层中间压紧下降[M]
ANDNOT W186.05  ; 进料爪上下层中间压紧下降[A]
LDNOT T0154  ; 进料爪上层中间压紧上升位延时
OR H0.09  ; 气缸保持（1保持）
ANDLD
OUT 106.04  ; 进料爪上下层中间压紧上升输出
LD TR0
LD W146.05  ; 进料爪上下层中间压紧下降[M]
OR W186.05  ; 进料爪上下层中间压紧下降[A]
OR 106.05  ; 进料爪上下层中间压紧下降输出
ANDLD
ANDNOT W146.04  ; 进料爪上下层中间压紧上升[M]
ANDNOT W186.04  ; 进料爪上下层中间压紧上升[A]
LD T0154  ; 进料爪上层中间压紧上升位延时
OR H0.09  ; 气缸保持（1保持）
ANDLD
OUT 106.05  ; 进料爪上下层中间压紧下降输出

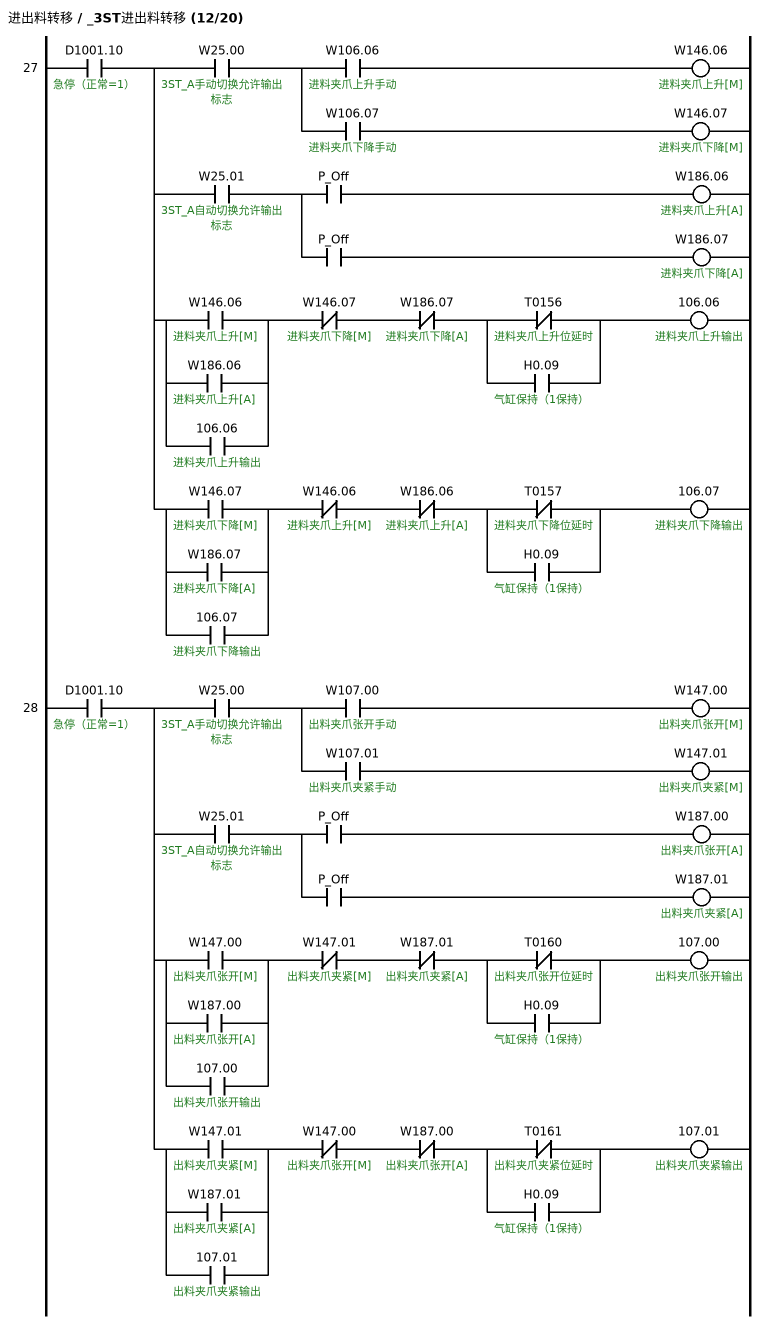
; rung 27
LD D1001.10  ; 急停（正常=1）
OUT TR0
AND W25.00  ; 3ST_A手动切换允许输出标志
OUT TR1
AND W106.06  ; 进料夹爪上升手动
OUT W146.06  ; 进料夹爪上升[M]
LD TR1
AND W106.07  ; 进料夹爪下降手动
OUT W146.07  ; 进料夹爪下降[M]
LD TR0
AND W25.01  ; 3ST_A自动切换允许输出标志
OUT TR1
AND P_Off
OUT W186.06  ; 进料夹爪上升[A]
LD TR1
AND P_Off
OUT W186.07  ; 进料夹爪下降[A]
LD TR0
LD W146.06  ; 进料夹爪上升[M]
OR W186.06  ; 进料夹爪上升[A]
OR 106.06  ; 进料夹爪上升输出
ANDLD
ANDNOT W146.07  ; 进料夹爪下降[M]
ANDNOT W186.07  ; 进料夹爪下降[A]
LDNOT T0156  ; 进料夹爪上升位延时
OR H0.09  ; 气缸保持（1保持）
ANDLD
OUT 106.06  ; 进料夹爪上升输出
LD TR0
LD W146.07  ; 进料夹爪下降[M]
OR W186.07  ; 进料夹爪下降[A]
OR 106.07  ; 进料夹爪下降输出
ANDLD
ANDNOT W146.06  ; 进料夹爪上升[M]
ANDNOT W186.06  ; 进料夹爪上升[A]
LDNOT T0157  ; 进料夹爪下降位延时
OR H0.09  ; 气缸保持（1保持）
ANDLD
OUT 106.07  ; 进料夹爪下降输出
; rung 28
LD D1001.10  ; 急停（正常=1）
OUT TR0
AND W25.00  ; 3ST_A手动切换允许输出标志
OUT TR1
AND W107.00  ; 出料夹爪张开手动
OUT W147.00  ; 出料夹爪张开[M]
LD TR1
AND W107.01  ; 出料夹爪夹紧手动
OUT W147.01  ; 出料夹爪夹紧[M]
LD TR0
AND W25.01  ; 3ST_A自动切换允许输出标志
OUT TR1
AND P_Off
OUT W187.00  ; 出料夹爪张开[A]
LD TR1
AND P_Off
OUT W187.01  ; 出料夹爪夹紧[A]
LD TR0
LD W147.00  ; 出料夹爪张开[M]
OR W187.00  ; 出料夹爪张开[A]
OR 107.00  ; 出料夹爪张开输出
ANDLD
ANDNOT W147.01  ; 出料夹爪夹紧[M]
ANDNOT W187.01  ; 出料夹爪夹紧[A]
LDNOT T0160  ; 出料夹爪张开位延时
OR H0.09  ; 气缸保持（1保持）
ANDLD
OUT 107.00  ; 出料夹爪张开输出
LD TR0
LD W147.01  ; 出料夹爪夹紧[M]
OR W187.01  ; 出料夹爪夹紧[A]
OR 107.01  ; 出料夹爪夹紧输出
ANDLD
ANDNOT W147.00  ; 出料夹爪张开[M]
ANDNOT W187.00  ; 出料夹爪张开[A]
LDNOT T0161  ; 出料夹爪夹紧位延时
OR H0.09  ; 气缸保持（1保持）
ANDLD
OUT 107.01  ; 出料夹爪夹紧输出

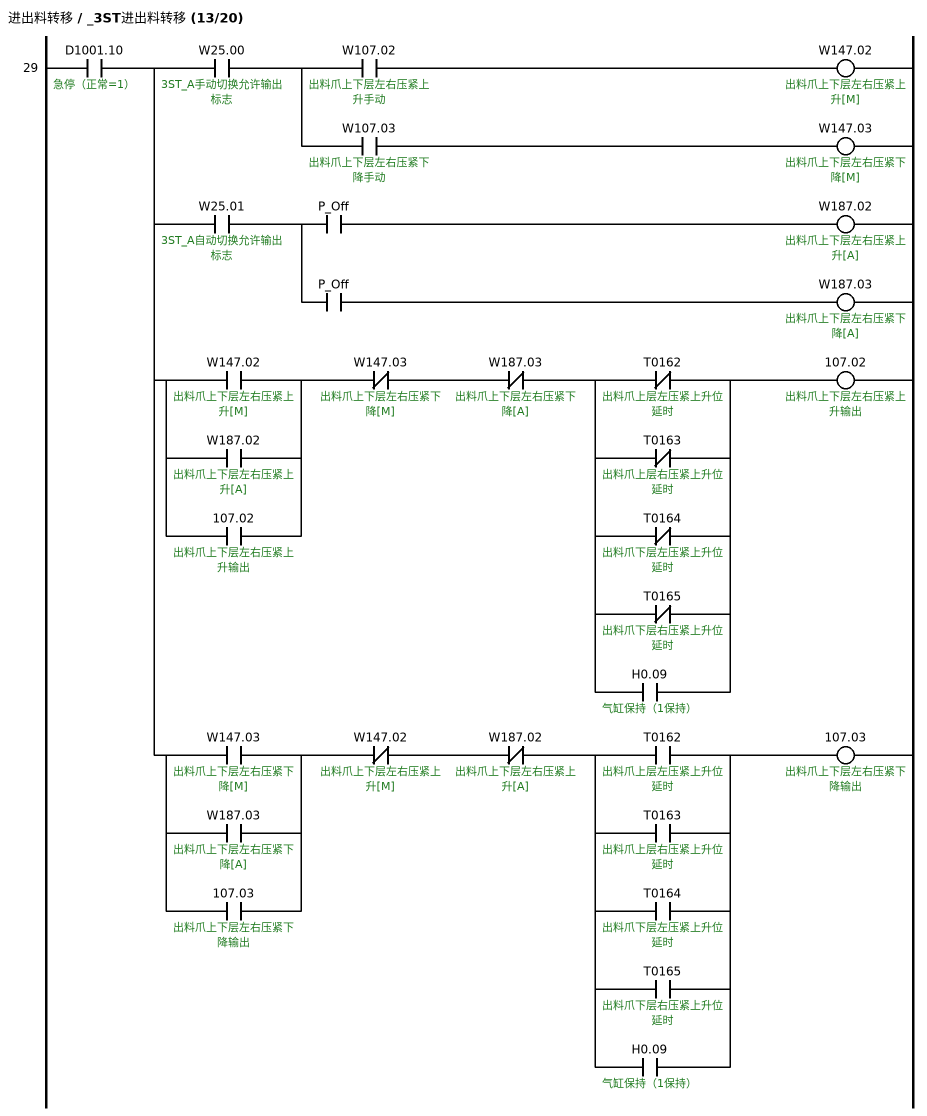
; rung 29
LD D1001.10  ; 急停（正常=1）
OUT TR0
AND W25.00  ; 3ST_A手动切换允许输出标志
OUT TR1
AND W107.02  ; 出料爪上下层左右压紧上升手动
OUT W147.02  ; 出料爪上下层左右压紧上升[M]
LD TR1
AND W107.03  ; 出料爪上下层左右压紧下降手动
OUT W147.03  ; 出料爪上下层左右压紧下降[M]
LD TR0
AND W25.01  ; 3ST_A自动切换允许输出标志
OUT TR1
AND P_Off
OUT W187.02  ; 出料爪上下层左右压紧上升[A]
LD TR1
AND P_Off
OUT W187.03  ; 出料爪上下层左右压紧下降[A]
LD TR0
LD W147.02  ; 出料爪上下层左右压紧上升[M]
OR W187.02  ; 出料爪上下层左右压紧上升[A]
OR 107.02  ; 出料爪上下层左右压紧上升输出
ANDLD
ANDNOT W147.03  ; 出料爪上下层左右压紧下降[M]
ANDNOT W187.03  ; 出料爪上下层左右压紧下降[A]
LDNOT T0162  ; 出料爪上层左压紧上升位延时
ORNOT T0163  ; 出料爪上层右压紧上升位延时
ORNOT T0164  ; 出料爪下层左压紧上升位延时
ORNOT T0165  ; 出料爪下层右压紧上升位延时
OR H0.09  ; 气缸保持（1保持）
ANDLD
OUT 107.02  ; 出料爪上下层左右压紧上升输出
LD TR0
LD W147.03  ; 出料爪上下层左右压紧下降[M]
OR W187.03  ; 出料爪上下层左右压紧下降[A]
OR 107.03  ; 出料爪上下层左右压紧下降输出
ANDLD
ANDNOT W147.02  ; 出料爪上下层左右压紧上升[M]
ANDNOT W187.02  ; 出料爪上下层左右压紧上升[A]
LD T0162  ; 出料爪上层左压紧上升位延时
OR T0163  ; 出料爪上层右压紧上升位延时
OR T0164  ; 出料爪下层左压紧上升位延时
OR T0165  ; 出料爪下层右压紧上升位延时
OR H0.09  ; 气缸保持（1保持）
ANDLD
OUT 107.03  ; 出料爪上下层左右压紧下降输出

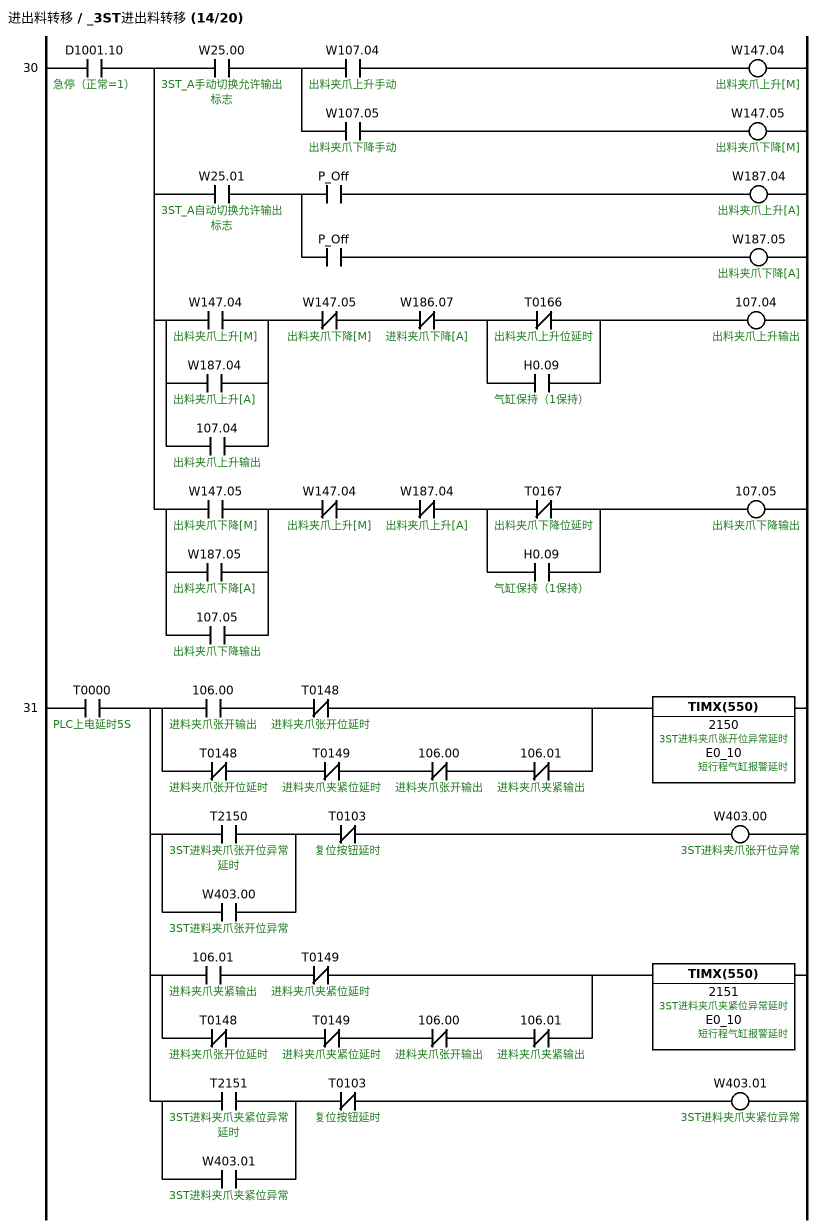
; rung 30
LD D1001.10  ; 急停（正常=1）
OUT TR0
AND W25.00  ; 3ST_A手动切换允许输出标志
OUT TR1
AND W107.04  ; 出料夹爪上升手动
OUT W147.04  ; 出料夹爪上升[M]
LD TR1
AND W107.05  ; 出料夹爪下降手动
OUT W147.05  ; 出料夹爪下降[M]
LD TR0
AND W25.01  ; 3ST_A自动切换允许输出标志
OUT TR1
AND P_Off
OUT W187.04  ; 出料夹爪上升[A]
LD TR1
AND P_Off
OUT W187.05  ; 出料夹爪下降[A]
LD TR0
LD W147.04  ; 出料夹爪上升[M]
OR W187.04  ; 出料夹爪上升[A]
OR 107.04  ; 出料夹爪上升输出
ANDLD
ANDNOT W147.05  ; 出料夹爪下降[M]
ANDNOT W186.07  ; 进料夹爪下降[A]
LDNOT T0166  ; 出料夹爪上升位延时
OR H0.09  ; 气缸保持（1保持）
ANDLD
OUT 107.04  ; 出料夹爪上升输出
LD TR0
LD W147.05  ; 出料夹爪下降[M]
OR W187.05  ; 出料夹爪下降[A]
OR 107.05  ; 出料夹爪下降输出
ANDLD
ANDNOT W147.04  ; 出料夹爪上升[M]
ANDNOT W187.04  ; 出料夹爪上升[A]
LDNOT T0167  ; 出料夹爪下降位延时
OR H0.09  ; 气缸保持（1保持）
ANDLD
OUT 107.05  ; 出料夹爪下降输出
; rung 31
LD T0000  ; PLC上电延时5S
OUT TR0
LD 106.00  ; 进料夹爪张开输出
ANDNOT T0148  ; 进料夹爪张开位延时
LDNOT T0148  ; 进料夹爪张开位延时
ANDNOT T0149  ; 进料夹爪夹紧位延时
ANDNOT 106.00  ; 进料夹爪张开输出
ANDNOT 106.01  ; 进料夹爪夹紧输出
ORLD
ANDLD
TIMX(550) 2150 E0_10  ; 短行程气缸报警延时, 3ST进料夹爪张开位异常延时
LD TR0
LD T2150  ; 3ST进料夹爪张开位异常延时
OR W403.00  ; 3ST进料夹爪张开位异常
ANDLD
ANDNOT T0103  ; 复位按钮延时
OUT W403.00  ; 3ST进料夹爪张开位异常
LD TR0
LD 106.01  ; 进料夹爪夹紧输出
ANDNOT T0149  ; 进料夹爪夹紧位延时
LDNOT T0148  ; 进料夹爪张开位延时
ANDNOT T0149  ; 进料夹爪夹紧位延时
ANDNOT 106.00  ; 进料夹爪张开输出
ANDNOT 106.01  ; 进料夹爪夹紧输出
ORLD
ANDLD
TIMX(550) 2151 E0_10  ; 短行程气缸报警延时, 3ST进料夹爪夹紧位异常延时
LD TR0
LD T2151  ; 3ST进料夹爪夹紧位异常延时
OR W403.01  ; 3ST进料夹爪夹紧位异常
ANDLD
ANDNOT T0103  ; 复位按钮延时
OUT W403.01  ; 3ST进料夹爪夹紧位异常

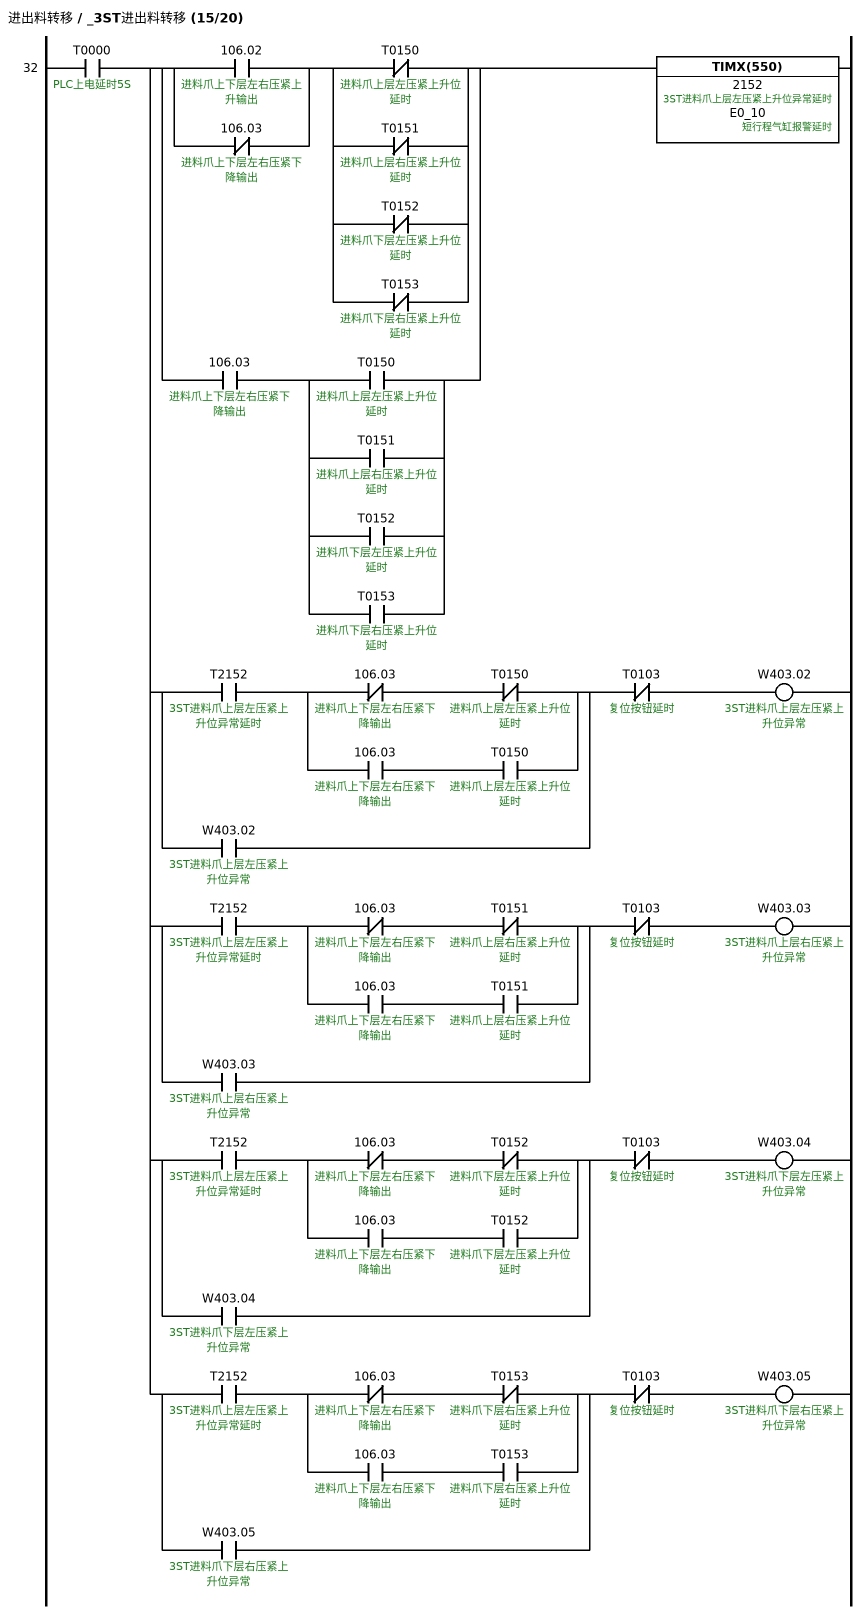
; rung 32
LD T0000  ; PLC上电延时5S
OUT TR0
LD 106.02  ; 进料爪上下层左右压紧上升输出
ORNOT 106.03  ; 进料爪上下层左右压紧下降输出
LDNOT T0150  ; 进料爪上层左压紧上升位延时
ORNOT T0151  ; 进料爪上层右压紧上升位延时
ORNOT T0152  ; 进料爪下层左压紧上升位延时
ORNOT T0153  ; 进料爪下层右压紧上升位延时
ANDLD
LD 106.03  ; 进料爪上下层左右压紧下降输出
LD T0150  ; 进料爪上层左压紧上升位延时
OR T0151  ; 进料爪上层右压紧上升位延时
OR T0152  ; 进料爪下层左压紧上升位延时
OR T0153  ; 进料爪下层右压紧上升位延时
ANDLD
ORLD
ANDLD
TIMX(550) 2152 E0_10  ; 短行程气缸报警延时, 3ST进料爪上层左压紧上升位异常延时
LD TR0
LD T2152  ; 3ST进料爪上层左压紧上升位异常延时
LDNOT 106.03  ; 进料爪上下层左右压紧下降输出
ANDNOT T0150  ; 进料爪上层左压紧上升位延时
LD 106.03  ; 进料爪上下层左右压紧下降输出
AND T0150  ; 进料爪上层左压紧上升位延时
ORLD
ANDLD
OR W403.02  ; 3ST进料爪上层左压紧上升位异常
ANDLD
ANDNOT T0103  ; 复位按钮延时
OUT W403.02  ; 3ST进料爪上层左压紧上升位异常
LD TR0
LD T2152  ; 3ST进料爪上层左压紧上升位异常延时
LDNOT 106.03  ; 进料爪上下层左右压紧下降输出
ANDNOT T0151  ; 进料爪上层右压紧上升位延时
LD 106.03  ; 进料爪上下层左右压紧下降输出
AND T0151  ; 进料爪上层右压紧上升位延时
ORLD
ANDLD
OR W403.03  ; 3ST进料爪上层右压紧上升位异常
ANDLD
ANDNOT T0103  ; 复位按钮延时
OUT W403.03  ; 3ST进料爪上层右压紧上升位异常
LD TR0
LD T2152  ; 3ST进料爪上层左压紧上升位异常延时
LDNOT 106.03  ; 进料爪上下层左右压紧下降输出
ANDNOT T0152  ; 进料爪下层左压紧上升位延时
LD 106.03  ; 进料爪上下层左右压紧下降输出
AND T0152  ; 进料爪下层左压紧上升位延时
ORLD
ANDLD
OR W403.04  ; 3ST进料爪下层左压紧上升位异常
ANDLD
ANDNOT T0103  ; 复位按钮延时
OUT W403.04  ; 3ST进料爪下层左压紧上升位异常
LD TR0
LD T2152  ; 3ST进料爪上层左压紧上升位异常延时
LDNOT 106.03  ; 进料爪上下层左右压紧下降输出
ANDNOT T0153  ; 进料爪下层右压紧上升位延时
LD 106.03  ; 进料爪上下层左右压紧下降输出
AND T0153  ; 进料爪下层右压紧上升位延时
ORLD
ANDLD
OR W403.05  ; 3ST进料爪下层右压紧上升位异常
ANDLD
ANDNOT T0103  ; 复位按钮延时
OUT W403.05  ; 3ST进料爪下层右压紧上升位异常

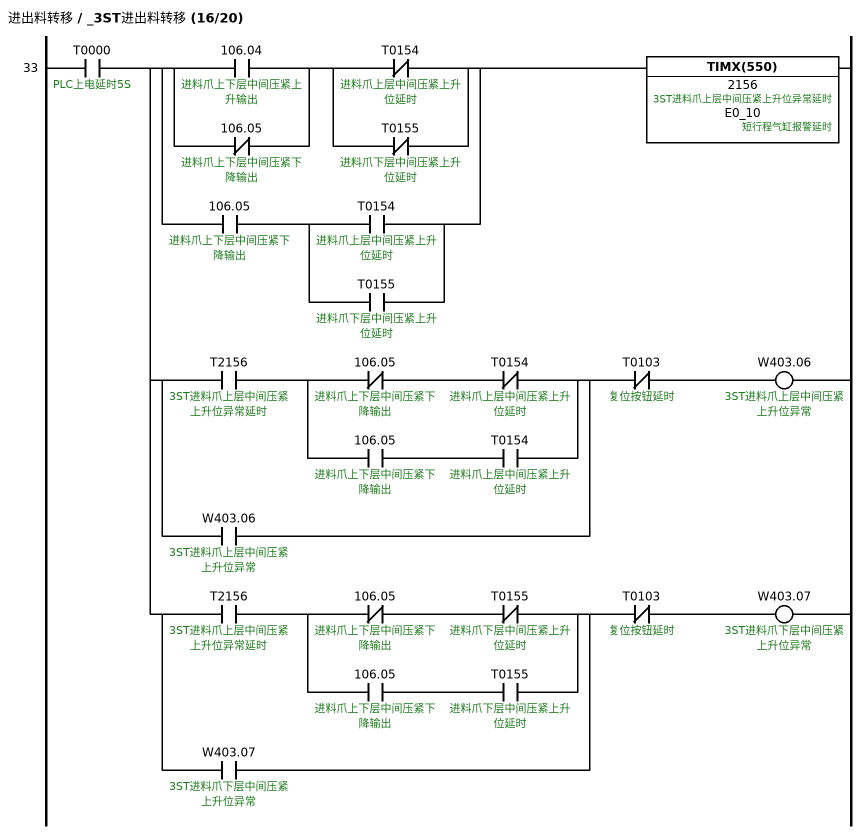
; rung 33
LD T0000  ; PLC上电延时5S
OUT TR0
LD 106.04  ; 进料爪上下层中间压紧上升输出
ORNOT 106.05  ; 进料爪上下层中间压紧下降输出
LDNOT T0154  ; 进料爪上层中间压紧上升位延时
ORNOT T0155  ; 进料爪下层中间压紧上升位延时
ANDLD
LD 106.05  ; 进料爪上下层中间压紧下降输出
LD T0154  ; 进料爪上层中间压紧上升位延时
OR T0155  ; 进料爪下层中间压紧上升位延时
ANDLD
ORLD
ANDLD
TIMX(550) 2156 E0_10  ; 短行程气缸报警延时, 3ST进料爪上层中间压紧上升位异常延时
LD TR0
LD T2156  ; 3ST进料爪上层中间压紧上升位异常延时
LDNOT 106.05  ; 进料爪上下层中间压紧下降输出
ANDNOT T0154  ; 进料爪上层中间压紧上升位延时
LD 106.05  ; 进料爪上下层中间压紧下降输出
AND T0154  ; 进料爪上层中间压紧上升位延时
ORLD
ANDLD
OR W403.06  ; 3ST进料爪上层中间压紧上升位异常
ANDLD
ANDNOT T0103  ; 复位按钮延时
OUT W403.06  ; 3ST进料爪上层中间压紧上升位异常
LD TR0
LD T2156  ; 3ST进料爪上层中间压紧上升位异常延时
LDNOT 106.05  ; 进料爪上下层中间压紧下降输出
ANDNOT T0155  ; 进料爪下层中间压紧上升位延时
LD 106.05  ; 进料爪上下层中间压紧下降输出
AND T0155  ; 进料爪下层中间压紧上升位延时
ORLD
ANDLD
OR W403.07  ; 3ST进料爪下层中间压紧上升位异常
ANDLD
ANDNOT T0103  ; 复位按钮延时
OUT W403.07  ; 3ST进料爪下层中间压紧上升位异常

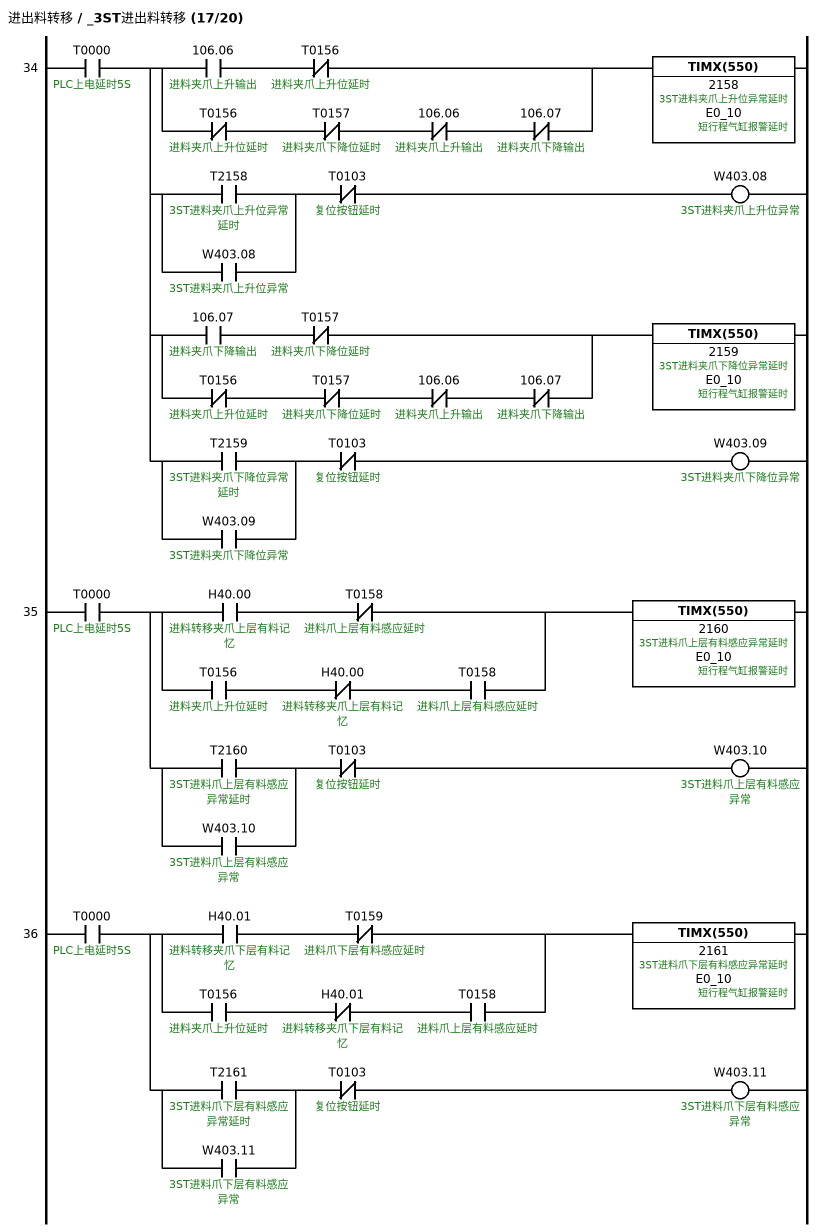
; rung 34
LD T0000  ; PLC上电延时5S
OUT TR0
LD 106.06  ; 进料夹爪上升输出
ANDNOT T0156  ; 进料夹爪上升位延时
LDNOT T0156  ; 进料夹爪上升位延时
ANDNOT T0157  ; 进料夹爪下降位延时
ANDNOT 106.06  ; 进料夹爪上升输出
ANDNOT 106.07  ; 进料夹爪下降输出
ORLD
ANDLD
TIMX(550) 2158 E0_10  ; 短行程气缸报警延时, 3ST进料夹爪上升位异常延时
LD TR0
LD T2158  ; 3ST进料夹爪上升位异常延时
OR W403.08  ; 3ST进料夹爪上升位异常
ANDLD
ANDNOT T0103  ; 复位按钮延时
OUT W403.08  ; 3ST进料夹爪上升位异常
LD TR0
LD 106.07  ; 进料夹爪下降输出
ANDNOT T0157  ; 进料夹爪下降位延时
LDNOT T0156  ; 进料夹爪上升位延时
ANDNOT T0157  ; 进料夹爪下降位延时
ANDNOT 106.06  ; 进料夹爪上升输出
ANDNOT 106.07  ; 进料夹爪下降输出
ORLD
ANDLD
TIMX(550) 2159 E0_10  ; 短行程气缸报警延时, 3ST进料夹爪下降位异常延时
LD TR0
LD T2159  ; 3ST进料夹爪下降位异常延时
OR W403.09  ; 3ST进料夹爪下降位异常
ANDLD
ANDNOT T0103  ; 复位按钮延时
OUT W403.09  ; 3ST进料夹爪下降位异常
; rung 35
LD T0000  ; PLC上电延时5S
OUT TR0
LD H40.00  ; 进料转移夹爪上层有料记忆
ANDNOT T0158  ; 进料爪上层有料感应延时
LD T0156  ; 进料夹爪上升位延时
ANDNOT H40.00  ; 进料转移夹爪上层有料记忆
AND T0158  ; 进料爪上层有料感应延时
ORLD
ANDLD
TIMX(550) 2160 E0_10  ; 短行程气缸报警延时, 3ST进料爪上层有料感应异常延时
LD TR0
LD T2160  ; 3ST进料爪上层有料感应异常延时
OR W403.10  ; 3ST进料爪上层有料感应异常
ANDLD
ANDNOT T0103  ; 复位按钮延时
OUT W403.10  ; 3ST进料爪上层有料感应异常
; rung 36
LD T0000  ; PLC上电延时5S
OUT TR0
LD H40.01  ; 进料转移夹爪下层有料记忆
ANDNOT T0159  ; 进料爪下层有料感应延时
LD T0156  ; 进料夹爪上升位延时
ANDNOT H40.01  ; 进料转移夹爪下层有料记忆
AND T0158  ; 进料爪上层有料感应延时
ORLD
ANDLD
TIMX(550) 2161 E0_10  ; 短行程气缸报警延时, 3ST进料爪下层有料感应异常延时
LD TR0
LD T2161  ; 3ST进料爪下层有料感应异常延时
OR W403.11  ; 3ST进料爪下层有料感应异常
ANDLD
ANDNOT T0103  ; 复位按钮延时
OUT W403.11  ; 3ST进料爪下层有料感应异常

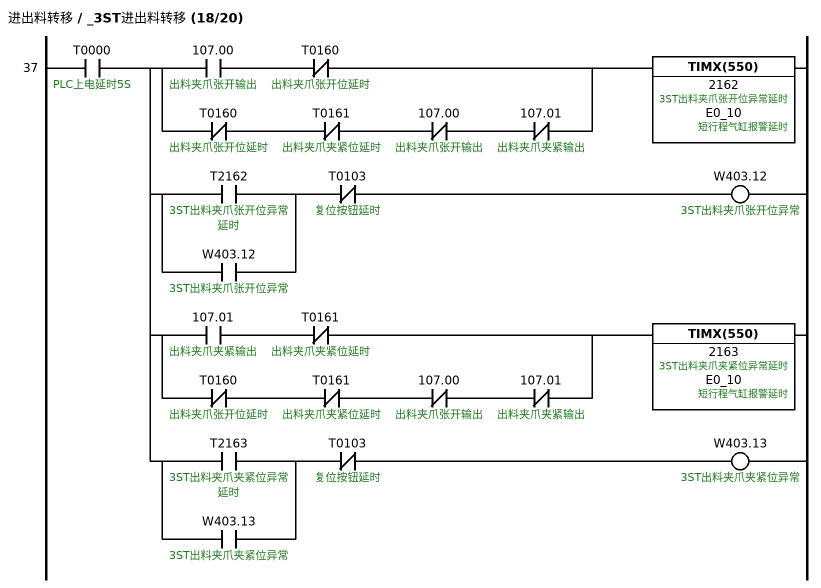
; rung 37
LD T0000  ; PLC上电延时5S
OUT TR0
LD 107.00  ; 出料夹爪张开输出
ANDNOT T0160  ; 出料夹爪张开位延时
LDNOT T0160  ; 出料夹爪张开位延时
ANDNOT T0161  ; 出料夹爪夹紧位延时
ANDNOT 107.00  ; 出料夹爪张开输出
ANDNOT 107.01  ; 出料夹爪夹紧输出
ORLD
ANDLD
TIMX(550) 2162 E0_10  ; 短行程气缸报警延时, 3ST出料夹爪张开位异常延时
LD TR0
LD T2162  ; 3ST出料夹爪张开位异常延时
OR W403.12  ; 3ST出料夹爪张开位异常
ANDLD
ANDNOT T0103  ; 复位按钮延时
OUT W403.12  ; 3ST出料夹爪张开位异常
LD TR0
LD 107.01  ; 出料夹爪夹紧输出
ANDNOT T0161  ; 出料夹爪夹紧位延时
LDNOT T0160  ; 出料夹爪张开位延时
ANDNOT T0161  ; 出料夹爪夹紧位延时
ANDNOT 107.00  ; 出料夹爪张开输出
ANDNOT 107.01  ; 出料夹爪夹紧输出
ORLD
ANDLD
TIMX(550) 2163 E0_10  ; 短行程气缸报警延时, 3ST出料夹爪夹紧位异常延时
LD TR0
LD T2163  ; 3ST出料夹爪夹紧位异常延时
OR W403.13  ; 3ST出料夹爪夹紧位异常
ANDLD
ANDNOT T0103  ; 复位按钮延时
OUT W403.13  ; 3ST出料夹爪夹紧位异常

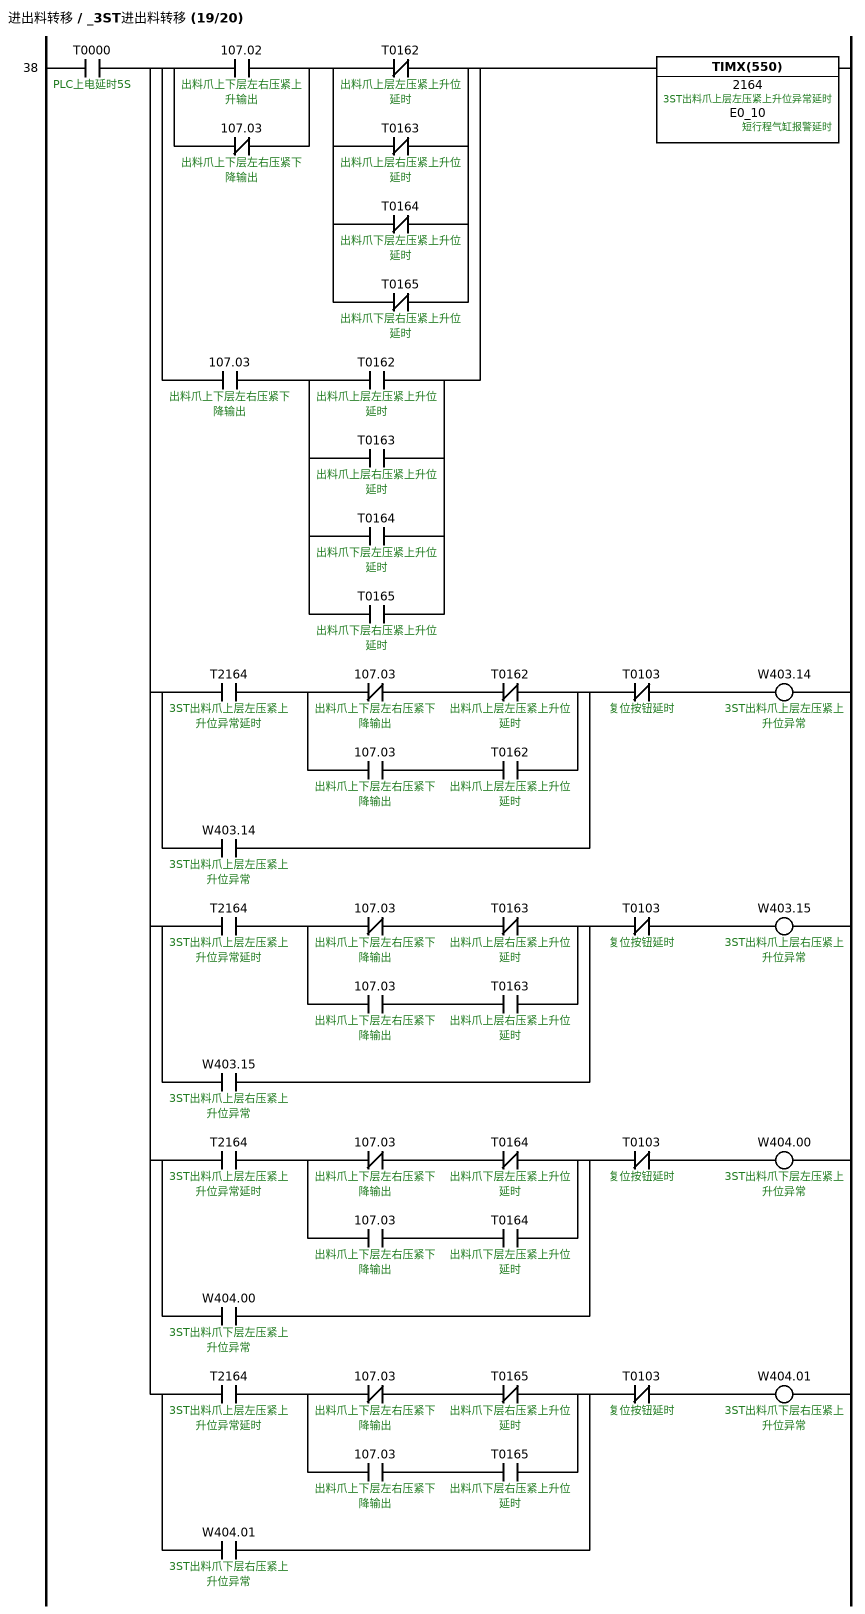
; rung 38
LD T0000  ; PLC上电延时5S
OUT TR0
LD 107.02  ; 出料爪上下层左右压紧上升输出
ORNOT 107.03  ; 出料爪上下层左右压紧下降输出
LDNOT T0162  ; 出料爪上层左压紧上升位延时
ORNOT T0163  ; 出料爪上层右压紧上升位延时
ORNOT T0164  ; 出料爪下层左压紧上升位延时
ORNOT T0165  ; 出料爪下层右压紧上升位延时
ANDLD
LD 107.03  ; 出料爪上下层左右压紧下降输出
LD T0162  ; 出料爪上层左压紧上升位延时
OR T0163  ; 出料爪上层右压紧上升位延时
OR T0164  ; 出料爪下层左压紧上升位延时
OR T0165  ; 出料爪下层右压紧上升位延时
ANDLD
ORLD
ANDLD
TIMX(550) 2164 E0_10  ; 短行程气缸报警延时, 3ST出料爪上层左压紧上升位异常延时
LD TR0
LD T2164  ; 3ST出料爪上层左压紧上升位异常延时
LDNOT 107.03  ; 出料爪上下层左右压紧下降输出
ANDNOT T0162  ; 出料爪上层左压紧上升位延时
LD 107.03  ; 出料爪上下层左右压紧下降输出
AND T0162  ; 出料爪上层左压紧上升位延时
ORLD
ANDLD
OR W403.14  ; 3ST出料爪上层左压紧上升位异常
ANDLD
ANDNOT T0103  ; 复位按钮延时
OUT W403.14  ; 3ST出料爪上层左压紧上升位异常
LD TR0
LD T2164  ; 3ST出料爪上层左压紧上升位异常延时
LDNOT 107.03  ; 出料爪上下层左右压紧下降输出
ANDNOT T0163  ; 出料爪上层右压紧上升位延时
LD 107.03  ; 出料爪上下层左右压紧下降输出
AND T0163  ; 出料爪上层右压紧上升位延时
ORLD
ANDLD
OR W403.15  ; 3ST出料爪上层右压紧上升位异常
ANDLD
ANDNOT T0103  ; 复位按钮延时
OUT W403.15  ; 3ST出料爪上层右压紧上升位异常
LD TR0
LD T2164  ; 3ST出料爪上层左压紧上升位异常延时
LDNOT 107.03  ; 出料爪上下层左右压紧下降输出
ANDNOT T0164  ; 出料爪下层左压紧上升位延时
LD 107.03  ; 出料爪上下层左右压紧下降输出
AND T0164  ; 出料爪下层左压紧上升位延时
ORLD
ANDLD
OR W404.00  ; 3ST出料爪下层左压紧上升位异常
ANDLD
ANDNOT T0103  ; 复位按钮延时
OUT W404.00  ; 3ST出料爪下层左压紧上升位异常
LD TR0
LD T2164  ; 3ST出料爪上层左压紧上升位异常延时
LDNOT 107.03  ; 出料爪上下层左右压紧下降输出
ANDNOT T0165  ; 出料爪下层右压紧上升位延时
LD 107.03  ; 出料爪上下层左右压紧下降输出
AND T0165  ; 出料爪下层右压紧上升位延时
ORLD
ANDLD
OR W404.01  ; 3ST出料爪下层右压紧上升位异常
ANDLD
ANDNOT T0103  ; 复位按钮延时
OUT W404.01  ; 3ST出料爪下层右压紧上升位异常

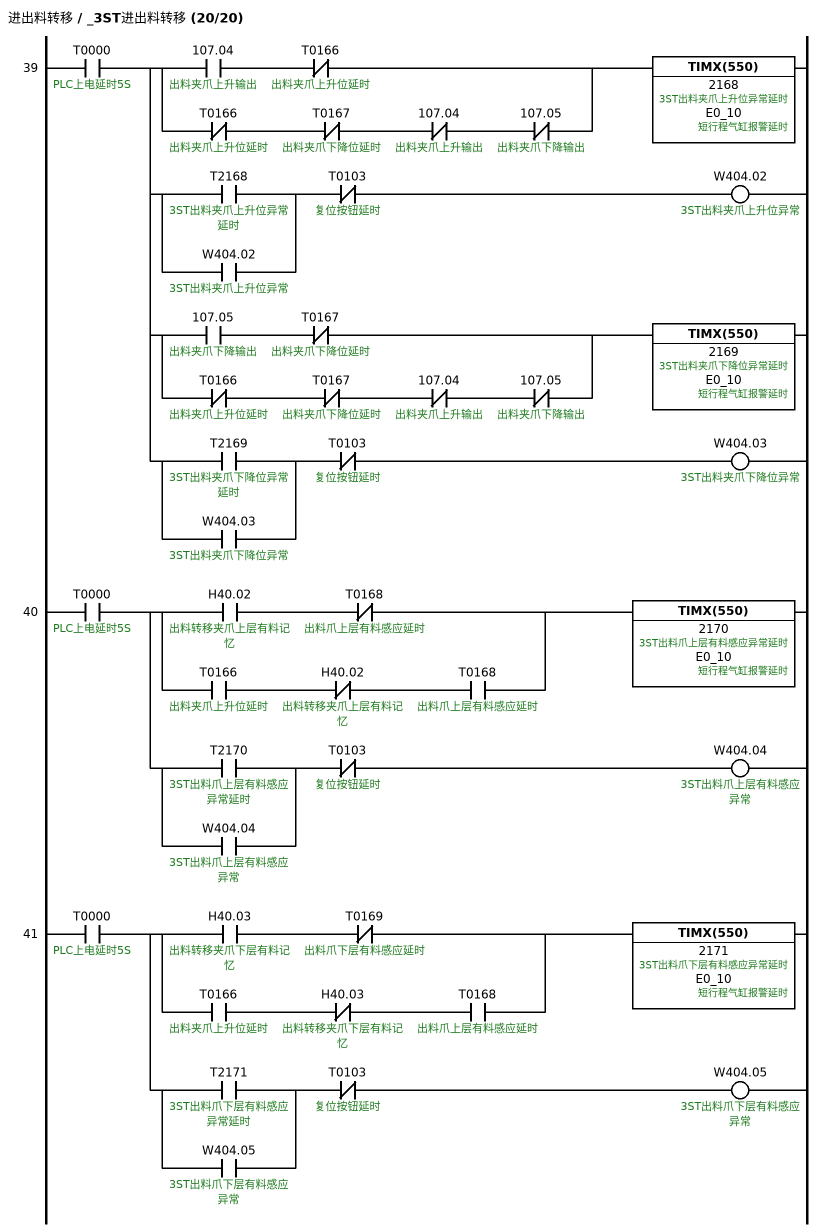
; rung 39
LD T0000  ; PLC上电延时5S
OUT TR0
LD 107.04  ; 出料夹爪上升输出
ANDNOT T0166  ; 出料夹爪上升位延时
LDNOT T0166  ; 出料夹爪上升位延时
ANDNOT T0167  ; 出料夹爪下降位延时
ANDNOT 107.04  ; 出料夹爪上升输出
ANDNOT 107.05  ; 出料夹爪下降输出
ORLD
ANDLD
TIMX(550) 2168 E0_10  ; 短行程气缸报警延时, 3ST出料夹爪上升位异常延时
LD TR0
LD T2168  ; 3ST出料夹爪上升位异常延时
OR W404.02  ; 3ST出料夹爪上升位异常
ANDLD
ANDNOT T0103  ; 复位按钮延时
OUT W404.02  ; 3ST出料夹爪上升位异常
LD TR0
LD 107.05  ; 出料夹爪下降输出
ANDNOT T0167  ; 出料夹爪下降位延时
LDNOT T0166  ; 出料夹爪上升位延时
ANDNOT T0167  ; 出料夹爪下降位延时
ANDNOT 107.04  ; 出料夹爪上升输出
ANDNOT 107.05  ; 出料夹爪下降输出
ORLD
ANDLD
TIMX(550) 2169 E0_10  ; 短行程气缸报警延时, 3ST出料夹爪下降位异常延时
LD TR0
LD T2169  ; 3ST出料夹爪下降位异常延时
OR W404.03  ; 3ST出料夹爪下降位异常
ANDLD
ANDNOT T0103  ; 复位按钮延时
OUT W404.03  ; 3ST出料夹爪下降位异常
; rung 40
LD T0000  ; PLC上电延时5S
OUT TR0
LD H40.02  ; 出料转移夹爪上层有料记忆
ANDNOT T0168  ; 出料爪上层有料感应延时
LD T0166  ; 出料夹爪上升位延时
ANDNOT H40.02  ; 出料转移夹爪上层有料记忆
AND T0168  ; 出料爪上层有料感应延时
ORLD
ANDLD
TIMX(550) 2170 E0_10  ; 短行程气缸报警延时, 3ST出料爪上层有料感应异常延时
LD TR0
LD T2170  ; 3ST出料爪上层有料感应异常延时
OR W404.04  ; 3ST出料爪上层有料感应异常
ANDLD
ANDNOT T0103  ; 复位按钮延时
OUT W404.04  ; 3ST出料爪上层有料感应异常
; rung 41
LD T0000  ; PLC上电延时5S
OUT TR0
LD H40.03  ; 出料转移夹爪下层有料记忆
ANDNOT T0169  ; 出料爪下层有料感应延时
LD T0166  ; 出料夹爪上升位延时
ANDNOT H40.03  ; 出料转移夹爪下层有料记忆
AND T0168  ; 出料爪上层有料感应延时
ORLD
ANDLD
TIMX(550) 2171 E0_10  ; 短行程气缸报警延时, 3ST出料爪下层有料感应异常延时
LD TR0
LD T2171  ; 3ST出料爪下层有料感应异常延时
OR W404.05  ; 3ST出料爪下层有料感应异常
ANDLD
ANDNOT T0103  ; 复位按钮延时
OUT W404.05  ; 3ST出料爪下层有料感应异常

### Section 复位

